# B&R Automation Studio project EasyLog
Automation Studio 4.12.3.127 SP; technology packages: mapp 5.24.1, mappCockpit 5.24.2, mappSafety 5.24.1, mappView 5.24.0

## Configuration C20

CPU 4PPC30.0702-21B, AutomationRuntime K4.93, Build 6.3.0, Safety 0.0, Vc V4.73.1

### Task classes (Cpu.sw)
```
Cyclic#2 (cycle 20000 us, tolerance 0 us):
  AsyncTask <- Async.AsyncTask.prg (AdditionalIncludeDirectories=\Logical\Async\AsyncCreation\ARM\, AdditionalLibraryDirectories=\Logical\Async\AsyncCreation\ARM\, AdditionalLibraries=AR)
  Example4 <- Example4.prg
Binaries: FWRules, arcoal, arsvcreg, TCData, arflatprv, mvLoader, udbdef, mCoWebSc, User, iomap, sysconf, Role, ashwd, arconfig, asfw, ashwac
Libraries: standard, runtime, astime, AsBrStr, sys_lib, ArEventLog, AsFifo, EasyLog, asiodiag, asioacc, SfDomDrv, SfDomVis, asepl, arssl, mpbase, MpSfDomMgr, aruser, fileio, asusb, astcp
```

### Hardware
```
4PPC30_0702_21B : 4PPC30.0702-21B v1.1.3.0
  Connector IF3:
    ActivateDevice = 1
    Mode = Manual
    InternetAddress = 10.10.10.100
    SubnetMask = 255.255.255.0
    InaPort = 11160
    ActivateSnmp = 2
  ConfigurationID = EasyLog_Config1
  TimerDeviceType = SWIOTIMER
  Cyclic1Duration = 10000
  Cyclic1Tolerance = 0
  Cyclic2Duration = 20000
  Cyclic2Tolerance = 0
  Cyclic3Duration = 50000
  Cyclic3Tolerance = 50000
  Cyclic4Duration = 100000
  Cyclic4Tolerance = 100000
  Cyclic5Duration = 200000
  Cyclic5Tolerance = 200000
  Cyclic6Duration = 500000
  Cyclic6Tolerance = 500000
  Cyclic7Duration = 1000000
  Cyclic7Tolerance = 1000000
  Cyclic7Stack = 65365
  Cyclic8Duration = 10000
  Cyclic8Tolerance = 30000000
  FileDevice1
  FileDeviceName1 = USER
  FileDevicePath1 = USER_PATH
  KeyMappingFile = VC\4PPC30_0702_21B1.dis
```

## Configuration Config1

CPU PC_any, AutomationRuntime I4.93, Build 6.3.0, Safety 0.0, Vc V4.73.1

### Task classes (Cpu.sw)
```
Cyclic#4:
  Program <- Program.prg
Binaries: FWRules, arcoal, arsvcreg, TCData, arflatprv, mvLoader, udbdef, mCoWebSc, User, iomap, sysconf, Role, ashwd, arconfig, asfw, ashwac
Libraries: AsIecCon, standard, runtime, astime, AsBrStr, DataObj, sys_lib, AsUSB, FileIO, AsSem, ArEventLog, AsARCfg, AsTCP, AsFifo, AsHttp, AsMem, EasyLog, asiodiag, asioacc, SfDomDrv, SfDomVis, asepl, arssl, mpbase, MpSfDomMgr, aruser
```

## Configuration ConfigNewC70

CPU 4PPC70.0573-20B, AutomationRuntime I4.93, Build 6.3.0, Vc V4.73.2

### Task classes (Cpu.sw)
```
Cyclic#2:
  Example4 <- Example4.prg
VcDataObjects: Visu1 <- Visu1.dob
Binaries: FWRules, arcoal, arsvcreg, TCData, arflatprv, mvLoader, udbdef, mCoWebSc, vcfile, arialbd, vcpdi855, vcbclass, vcnet, vcdsloc, Visu103, vccovl, vcptelo, vcshared, vcrt, vcpkat, vcpk, Visu101, vccbtn, vcmgr, Visu102, vctcal, vcalarm, vcpdsw, arial, vcgclass, vcpdvnc, vcpdihd, vcfntttf, vccstr, vcpdi815, vcpfppc7, vcdsint, User, iomap, sysconf, Role, ashwd, arconfig, asfw, ashwac
Libraries: EasyLog, AsBrStr, ArEventLog, astcp, asusb, astime, fileio, asiodiag, standard, asioacc, SfDomDrv, sys_lib, SfDomVis, asepl, runtime, arssl, mpbase, MpSfDomMgr, aruser, dataobj, vcresman
```

### Hardware
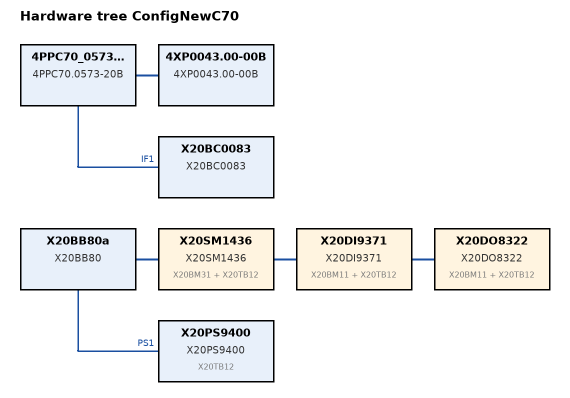
```
4PPC70_0573_20B : 4PPC70.0573-20B v1.5.4.0
  Connector IF2:
    ActivateDevice = 1
    Vnc1
    VncVcObjectName1 = Visu1
    VncKeyMappingFile1 = VC\PS2-Keyboard.dis
  ConfigurationID = EasyLog_ConfigNewC70
  UserPartitionSize = 0
  Cyclic1Tolerance = 0
  Cyclic2Tolerance = 0
  Cyclic7Stack = 65365
  FileDevice1
  FileDeviceName1 = USER
  FileDevicePath1 = USER_PATH
  VcObjectName = Visu1
  KeyMappingFile = VC\4PPC70_0573_20B.dis
4XP0043.00-00B : 4XP0043.00-00B v2.1.0.0  [X2X1 -> 4PPC70_0573_20B.IF5 [Cable Type=X2XCable, Length=10, Version=1.0.0.3]]
  Supervision = off
X20BB80a : X20BB80 v1.1.0.0
X20BC0083 : X20BC0083 v2.14.0.0  [PLK1 -> 4PPC70_0573_20B.IF1 (NodeNumber=1) [Cable Type=PowerlinkCable, Length=10, Version=1.0.0.3]; SL -> X20BB80a.SL1]
  Supervision = off
X20BM11a : X20BM11 v1.1.0.0  [X2X1 -> X20BM31a.X2X2]
X20BM11b : X20BM11 v1.1.0.0  [X2X1 -> X20BM11a.X2X2]
X20BM31a : X20BM31 v1.1.0.0  [X2X1 -> X20BB80a.IF1]
X20DI9371 : X20DI9371 v1.4.0.0  [SS1 -> X20TB12c.SS; SL -> X20BM11a.SL1]
  Supervision = off
X20DO8322 : X20DO8322 v1.5.0.0  [SS1 -> X20TB12d.SS; SL -> X20BM11b.SL1]
  Supervision = off
X20PS9400 : X20PS9400 v1.8.0.0  [SS1 -> X20TB12b.SS; PS -> X20BB80a.PS1]
  Supervision = off
X20SM1436 : X20SM1436 v2.3.0.0  [SS1 -> X20TB12a.SS; SL -> X20BM31a.SL1]
  FunctionModel = Standard
  Supervision = off
X20TB12a : X20TB12 v1.0.0.0
X20TB12b : X20TB12 v1.0.0.0
X20TB12c : X20TB12 v1.0.0.0
X20TB12d : X20TB12 v1.0.0.0
```

## Configuration Dinamic_Intel

CPU X20CP1686X, AutomationRuntime 6.0.2, Build 11.3.0, Vc 6.0.0

### Task classes (Cpu.sw)
```
Cyclic#4:
  Example1 <- Example1.prg
  Example2 <- Example2.prg
  Example3 <- Example3.prg
Libraries: EasyLog, runtime, ArEventLog, AsBrStr, sys_lib, standard
```

### Hardware
```
X20CP1686X : X20CP1686X v1.8.2.0
  FileDevice1
  FileDeviceName1 = USER
  FileDevicePath1 = USER_PATH
```

## Configuration Dynamic_ARM

CPU 4PPC30.043F-21B, AutomationRuntime 6.0.2, Build 11.3.0, Vc 6.0.0

### Task classes (Cpu.sw)
```
Cyclic#2 (cycle 20000 us, tolerance 20000 us):
  Example1 <- Example1.prg
  Example2 <- Example2.prg
  Example3 <- Example3.prg
Libraries: operator, runtime, AsIecCon, astime, EasyLog, ArEventLog, AsBrStr, sys_lib, standard
```

### Task classes (Cpu.sw)
```
Cyclic#3 (cycle 50000 us, tolerance 50000 us):
  Example2 <- Example2.prg
Cyclic#4 (cycle 100000 us, tolerance 100000 us):
  Example1 <- Example1.prg
Binaries: FWRules, TCData, mvLoader, udbdef, mCoWebSc, User, iomap, sysconf, Role, ashwd, arconfig, asfw, ashwac, arcoal, arsvcreg, arflatprv
Libraries: standard, runtime, EasyLog, asstring, astime, AsBrStr, sys_lib, ArEventLog, AsFifo, SfDomDrv, SfDomVis, MpSfDomMgr, AsIecCon, AsMem, DataObj, AsARCfg, AsSem, AsHttp
```

### Hardware
```
4PPC30_043F_21B : 4PPC30.043F-21B v1.1.4.0
  Connector IF3:
    ActivateDevice = 1
  ConfigurationID = EasyLog6_Dynamic_ARM
  TimerDeviceType = SWIOTIMER
  Cyclic1Duration = 10000
  Cyclic1Tolerance = 10000
  Cyclic2Duration = 20000
  Cyclic2Tolerance = 20000
  Cyclic3Duration = 50000
  Cyclic3Tolerance = 50000
  Cyclic4Duration = 100000
  Cyclic4Tolerance = 100000
  Cyclic5Duration = 200000
  Cyclic5Tolerance = 200000
  Cyclic6Duration = 500000
  Cyclic6Tolerance = 500000
  Cyclic7Duration = 1000000
  Cyclic7Tolerance = 1000000
  Cyclic8Duration = 10000
  Cyclic8Tolerance = 30000000
  FileDevice1
  FileDeviceName1 = USER
  FileDevicePath1 = USER_PATH
  KeyMappingFile = VC\4PPC30_043F_21B.dis
```

## Configuration Dynamic_ARM_2

CPU 4PPC30.043F-21B, AutomationRuntime K4.93, Build 6.3.0, Vc V4.73.2

### Task classes (Cpu.sw)
```
Cyclic#2 (cycle 20000 us, tolerance 20000 us):
  Example1 <- Example1.prg
  Example2 <- Example2.prg
  Example3 <- Example3.prg
Binaries: arsvcreg, udbdef, TCData, arflatprv, arcoal, mvLoader, FWRules, mCoWebSc, ashwac, User, sysconf, iomap, asfw, arconfig, ashwd, Role
Libraries: EasyLog, runtime, AsBrStr, sys_lib, ArEventLog, standard, astime, AsFifo, mpbase, arssl, SfDomVis, asiodiag, asioacc, aruser, fileio, SfDomDrv, asepl, MpSfDomMgr, asusb, astcp
```

### Hardware
```
4PPC30_043F_21B : 4PPC30.043F-21B v1.1.3.0
  Connector IF3:
    ActivateDevice = 1
  ConfigurationID = EasyLog_Dynamic_ARM_2
  TimerDeviceType = SWIOTIMER
  Cyclic1Duration = 10000
  Cyclic1Tolerance = 10000
  Cyclic2Duration = 20000
  Cyclic2Tolerance = 20000
  Cyclic3Duration = 50000
  Cyclic3Tolerance = 50000
  Cyclic4Duration = 100000
  Cyclic4Tolerance = 100000
  Cyclic5Duration = 200000
  Cyclic5Tolerance = 200000
  Cyclic6Duration = 500000
  Cyclic6Tolerance = 500000
  Cyclic7Duration = 1000000
  Cyclic7Tolerance = 1000000
  Cyclic8Duration = 10000
  Cyclic8Tolerance = 30000000
  FileDevice1
  FileDeviceName1 = USER
  FileDevicePath1 = USER_PATH
  KeyMappingFile = VC\4PPC30_043F_21B.dis
```

## Configuration Dynamic_Intel

CPU PC_any, AutomationRuntime K4.93, Build 6.3.0, Safety 0.0, Vc V4.73.1

CPU X20CP1586, AutomationRuntime H4.93, Build 6.3.0, Safety 0.0, Vc V4.73.1

### Task classes (Cpu.sw)
```
Cyclic#3:
  Example2 <- Example2.prg
Cyclic#4:
  Example1 <- Example1.prg
Binaries: FWRules, arcoal, arsvcreg, TCData, arflatprv, mvLoader, udbdef, mCoWebSc, User, iomap, sysconf, Role, ashwd, arconfig, asfw, ashwac
Libraries: standard, runtime, astime, AsBrStr, sys_lib, ArEventLog, AsFifo, asiodiag, asioacc, SfDomDrv, SfDomVis, asepl, arssl, mpbase, MpSfDomMgr, aruser, EasyLog, asstring
```

### Task classes (Cpu.sw)
```
Cyclic#2 (cycle 100000 us, tolerance 100000 us):
  Example1 <- Example1.prg
  Example2 <- Example2.prg
  Example3 <- Example3.prg
Binaries: FWRules, arcoal, arsvcreg, TCData, arflatprv, mvLoader, udbdef, mCoWebSc, User, iomap, sysconf, Role, ashwd, arconfig, asfw, ashwac
Libraries: standard, runtime, astime, AsBrStr, sys_lib, ArEventLog, AsFifo, EasyLog, asiodiag, asioacc, SfDomDrv, SfDomVis, asepl, arssl, mpbase, MpSfDomMgr, aruser, fileio, asusb, astcp
```

### Hardware
```
X20CP1586 : X20CP1586 v1.11.0.0
  Connector IF1:
    ActivateIna = 0
  Connector IF2:
    ActivateDevice = 1
    InaPort = 11160
  ConfigurationID = EasyLog_Config1
  Cyclic1Duration = 20000
  Cyclic1Tolerance = 0
  Cyclic1Stack = 522920
  Cyclic2Duration = 100000
  Cyclic2Tolerance = 100000
  FileDevice1
  FileDeviceName1 = USER
  FileDevicePath1 = USER_PATH
```

## Configuration ETA_Light

CPU 4PPC70.0573-20B, AutomationRuntime I4.93, Build 6.3.0, Safety 0.0, Vc V4.73.1

### Task classes (Cpu.sw)
```
Cyclic#2:
  Example4 <- Example4.prg
  AsyncTask <- Async.AsyncTask.prg (AdditionalIncludeDirectories=\Logical\Async\AsyncCreation\ARM\, AdditionalLibraryDirectories=\Logical\Async\AsyncCreation\ARM\, AdditionalLibraries=AR)
Binaries: FWRules, arcoal, arsvcreg, TCData, arflatprv, mvLoader, udbdef, mCoWebSc, User, iomap, sysconf, Role, ashwd, arconfig, asfw, ashwac
Libraries: standard, runtime, astime, AsBrStr, sys_lib, ArEventLog, AsFifo, EasyLog, asiodiag, asioacc, SfDomDrv, SfDomVis, asepl, arssl, mpbase, MpSfDomMgr, aruser, fileio, asusb, astcp
```

### Hardware
```
4PPC70_0573_20B : 4PPC70.0573-20B v1.5.4.0
  Connector IF2:
    ActivateDevice = 1
    Mode = Manual
    InternetAddress = 10.10.10.11
    SubnetMask = 255.255.255.0
    InaPort = 11160
    ActivateSnmp = 2
    DeviceParam = /EDDN=cpsw
  ConfigurationID = EasyLog_Config1
  Cyclic2Tolerance = 0
  Cyclic2Stack = 65365
  Cyclic7Stack = 65365
  FileDevice1
  FileDeviceName1 = USER
  FileDevicePath1 = USER_PATH
  KeyMappingFile = VC\4PPC70_0573_20B.dis
```

## Configuration Static_ARM

CPU X20CP0410, AutomationRuntime K4.93, Build 6.3.0, Safety 0.0, Vc V4.73.1

### Task classes (Cpu.sw)
```
Cyclic#3 (cycle 50000 us, tolerance 50000 us):
  Example2 <- Example2.prg
Cyclic#4 (cycle 100000 us, tolerance 100000 us):
  Example1 <- Example1.prg
Binaries: FWRules, arcoal, arsvcreg, TCData, arflatprv, mvLoader, udbdef, mCoWebSc, User, iomap, sysconf, Role, ashwd, arconfig, asfw, ashwac
Libraries: standard, runtime, astime, AsBrStr, sys_lib, ArEventLog, AsFifo, EasyLog, asiodiag, asioacc, SfDomDrv, SfDomVis, asepl, arssl, mpbase, MpSfDomMgr, aruser, AsIecCon, AsMem, DataObj, FileIO, AsARCfg, AsSem, AsHttp, AsUSB, AsTCP
```

### Hardware
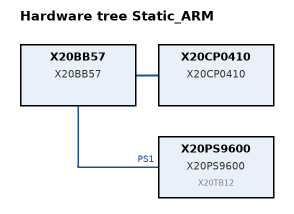
```
X20BB57 : X20BB57 v1.2.0.0
X20CP0410 : X20CP0410 v1.6.0.0  [SL -> X20BB57.SL1]
  Connector IF2:
    ActivateDevice = 1
    InaPort = 11160
  ConfigurationID = EasyLog_Config1
  TimerDeviceType = SWIOTIMER
  Cyclic1Duration = 10000
  Cyclic1Tolerance = 10000
  Cyclic2Duration = 20000
  Cyclic2Tolerance = 20000
  Cyclic3Duration = 50000
  Cyclic3Tolerance = 50000
  Cyclic4Duration = 100000
  Cyclic4Tolerance = 100000
  Cyclic5Duration = 200000
  Cyclic5Tolerance = 200000
  Cyclic6Duration = 500000
  Cyclic6Tolerance = 500000
  Cyclic7Duration = 1000000
  Cyclic7Tolerance = 1000000
  Cyclic8Duration = 10000
  Cyclic8Tolerance = 30000000
  FileDevice1
  FileDeviceName1 = USER
  FileDevicePath1 = USER_PATH
X20PS9600 : X20PS9600 v1.6.1.0  [PS -> X20BB57.PS1; SS1 -> X20TB12.SS]
X20TB12 : X20TB12 v1.0.0.0
```

## Configuration Static_Intel

CPU PC_any, AutomationRuntime K4.93, Build 6.3.0, Safety 0.0, Vc V4.73.1

### Task classes (Cpu.sw)
```
Cyclic#3:
  Example2 <- Example2.prg
Cyclic#4:
  Example1 <- Example1.prg
Binaries: FWRules, arcoal, arsvcreg, TCData, arflatprv, mvLoader, udbdef, mCoWebSc, User, iomap, sysconf, Role, ashwd, arconfig, asfw, ashwac
Libraries: standard, runtime, astime, AsBrStr, sys_lib, ArEventLog, AsFifo, EasyLog, asiodiag, asioacc, SfDomDrv, SfDomVis, asepl, arssl, mpbase, MpSfDomMgr, aruser
```

## Logical view

Binary libraries used (declarations not repeated): operator, runtime, AsIecCon, astime, ArEventLog, AsBrStr, sys_lib, standard, AsFifo

### Package Logical/Libraries - Global libraries

### Library Logical/Libraries/EasyLog (ANSIC, version 1.00.0)
Depends on: ArEventLog, AsBrStr, sys_lib

#### EasyLog.fun
```iecst
FUNCTION EasyLog : DINT (*Status returned by the function. Status <> ERR_OK should be checked*)
	VAR_INPUT
		Execute : BOOL; (*Input to add a message in the logger. Every cycle with TRUE in this input will insert a logger message. *) (* *) (*#PAR*)
		LoggerName : STRING[10]; (*String with the name of the Logger. Max Lenght 10 characters.*) (* *) (*#PAR*)
		LogLevel : USINT; (*Severity of the error. Coud be arEVENTLOG_SEVERITY_SUCCESS, arEVENTLOG_SEVERITY_INFO,  arEVENTLOG_SEVERITY_WARNING or arEVENTLOG_SEVERITY_ERROR*) (* *) (*#PAR*)
		ErrorNumber : UINT; (*Number of the error or information to insert*) (* *) (*#PAR*)
		Message : STRING[256]; (*String that specify the message to insert in the logger. Max lenght 256 characters*) (* *) (*#PAR*)
	END_VAR
END_FUNCTION
```

#### Logger.h
```c
#ifndef LOGGER_H
#define LOGGER_H

#include <stdlib.h>
#include "AsBrStr.h"
#include <cstring>
#include <string>

extern "C"
{
  long int EasyLog(plcbit Execute, plcstring* LoggerName, unsigned char LogLevel, unsigned short ErrorNumber, plcstring* Message);
}

#endif // LOGGER_H
```

#### EasyLog.cpp
```cpp
#include "Logger.h"
#include "EasyLog.h"
#include "LoggerInternal.hpp"

//extern "C" {
long int EasyLog(plcbit Execute, plcstring* LoggerName, unsigned char LogLevel, unsigned short ErrorNumber, plcstring* Message)
{
	Logger& logger = Logger::getInstance();
	return logger.EasyLogInternal(Execute, LoggerName, LogLevel, ErrorNumber, Message);
}
//}
```

#### LoggerInternal.hpp
```cpp
#ifndef LOGGERINTERNAL_H
#define LOGGERINTERNAL_H

#include "ArEventLog.h"
#include <stdlib.h>
#include "AsBrStr.h"
#include "runtime.h"
#include "sys_lib.h"
#include <iostream>
#include <cstring>
#include <string>
#include <queue>
#include <map>
#include "rtk.h"

struct LoggerEntry_type
{
	unsigned char LogLevel;
	long int ErrorNumber;
	char AsciiData[257];
};

struct LoggerHandler_type
{
	signed long ErrorInternal;
	char LoggerName[11];
	unsigned long pLoggerQueue;
	struct LoggerEntry_type LogEntry;
	unsigned long LogIdent;
	struct ArEventLogCreate ArEventLogCreate_0;
	RTK_TASK_H TaskHandler;
	bool CreatingLogger;
	bool CreateLogger;
};

class Logger {
public:
    static Logger& getInstance();
	long int EasyLogInternal(plcbit Execute, plcstring* LoggerName, unsigned char LogLevel, unsigned short ErrorNumber, plcstring* Message);

private:
    Logger() = default;
    ~Logger() = default;
    Logger(const Logger&) = delete;
    Logger& operator=(const Logger&) = delete;

	//Headers of the functions
    unsigned long SearchMap(unsigned long inst);
    long int UserLogEnqueue(unsigned char LogLevel, unsigned short ErrorNumber, unsigned long pAsciiData, unsigned long pLoggerName, unsigned long pHandler);
    long int UserLogWrite(unsigned long pHandler, bool fromAsync);
    long int UserLogCreateLog(unsigned long pHandler);
    long int UserLogGetIdent(unsigned long pHandler);
    static void CreateNewLoggerAsync(void* Params);

};

#endif // LOGGERINTERNAL_H
```

#### EasyLogInternal.cpp
```cpp
#include "LoggerInternal.hpp"
#include <cstdlib>
#include <cstring>

	/* Internal Data Map
	 * This map is used to store and retrieve the internal state for each instance, allowing
	 * for the management of multiple instances within the system. Related a Handler with all the information
	 * with one logger name given as a string */
std::map<std::string, unsigned long> internalMap;

	//Functions to get ident and write. As long as this functions have syncronous
	// execution does not have any sense save one copy of each function in the handler
struct ArEventLogGetIdent ArEventLogGetIdent_0;
struct ArEventLogWrite ArEventLogWrite_0;

Logger& Logger::getInstance() {
	static Logger instance;
	return instance;
}

/**
 * Retrieves or creates the internal data structure for the given instance.
 *
 * This function checks if an internal data structure for the provided instance
 * exists in the internal map. If it does not, it initializes a new internal
 * structure and stores it in the map.
 */
unsigned long Logger::SearchMap(unsigned long inst)
{
	//Retrieve the logger name
	std::string loggerName((char*)inst);
	std::map<std::string, unsigned long>::iterator it;

	//Search the Handler with the logger name
	it = internalMap.find(loggerName);

	//If it is not found, create a new Handler to insert to the map with the new logger name
	if (it == internalMap.end())
	{
		//Local instance of the handler
		struct LoggerHandler_type newHandler = {0};
		newHandler.LoggerName[11] = {0};
		std::strncpy(newHandler.LoggerName, loggerName.c_str(), sizeof(newHandler.LoggerName) - 1);

		//Create a local instance of queue, allocate it in memory and
		//achieve the pointer to that queue to store it in the local handler
		std::queue<LoggerEntry_type>* localLoggerQueue = (std::queue<LoggerEntry_type>*)malloc(sizeof(std::queue<LoggerEntry_type>));
		new(localLoggerQueue) std::queue<LoggerEntry_type>();
		newHandler.pLoggerQueue = reinterpret_cast<unsigned long>(localLoggerQueue);

		//Allocate the Handler in memory and save the local instance)
		LoggerHandler_type* savedInstance = (LoggerHandler_type*)malloc(sizeof(LoggerHandler_type));

		//Copy the local instance to the saved memory
		brsmemcpy((UDINT)savedInstance, (UDINT)&newHandler, sizeof(LoggerHandler_type));

		//Store the pointer of the saved instance
		unsigned long pHandler = reinterpret_cast<unsigned int>(savedInstance);

		//Save the new instance in the map and return it
		internalMap[loggerName] = pHandler;
		return internalMap[loggerName];
	}
	//If it is found return the Handler
	else
	{
		return it->second;
	}
}

/* Function to execute when is necessary a log insertion.
	It will be enqueued in a Queue until the UserLogWrite inserts the messages in the logger*/
long int Logger::UserLogEnqueue(unsigned char LogLevel, unsigned short ErrorNumber, unsigned long pAsciiData, unsigned long pLoggerName, unsigned long pHandler)
{
	//Initial status
	long int Status = ERR_OK;

	//Retrieve the Handler and its queue through its pointers
	struct LoggerHandler_type* Handler = reinterpret_cast<LoggerHandler_type*>(pHandler);
	std::queue<LoggerEntry_type>* queue = reinterpret_cast<std::queue<LoggerEntry_type>*>(Handler->pLoggerQueue);

	//Check not null pointers
	if (pHandler == 0 || Handler->pLoggerQueue == 0)
	{
		Status = ERR_BUR_ILLBPTR;
	}
	else
	{
		//Create a new entry type with the external information
		LoggerEntry_type newEntry;
		newEntry.LogLevel = LogLevel;
		newEntry.ErrorNumber = ErrorNumber;
		brsmemcpy((UDINT)&newEntry.AsciiData, pAsciiData, sizeof(newEntry.AsciiData));

		//Push that entry in the queue
		queue->push(newEntry);
	}

	return Status;
}

//Function to execute asyncronously with the Logger name to insert
// the messages in the logger that has been inserted with the UserLogEnqueue function
long int Logger::UserLogWrite(unsigned long pHandler, bool fromAsync)
{
	//Initialize the Status
	long int Status = ERR_OK;

	//Retrieve the Handler and its queue through its pointers
	struct LoggerHandler_type* Handler = reinterpret_cast<LoggerHandler_type*>(pHandler);
	std::queue<LoggerEntry_type>* queue = reinterpret_cast<std::queue<LoggerEntry_type>*>(Handler->pLoggerQueue);

	//Check not null pointers
	if (pHandler == 0 || Handler->pLoggerQueue == 0)
	{
		Status = ERR_BUR_ILLBPTR;
	}
	else
	{
		//If it is not busy the creation of the logger
		if (!Handler->CreatingLogger || fromAsync)
		{
			//Check if it is necessary to write the log
			if (queue->size() > 0 && Handler->LogIdent != 0)
			{
				int elements = queue->size();
				for (int i = 0; i < elements; i++)
				{
					// Put the first entry in the Handler
					Handler->LogEntry = queue->front();

					//Set the parameters of the write function
					ArEventLogWrite_0.Execute = 1;
					ArEventLogWrite_0.AddDataFormat = arEVENTLOG_ADDFORMAT_TEXT;
					ArEventLogWrite_0.AddDataSize = brsstrlen((UDINT)&Handler->LogEntry.AsciiData) + 1;
					ArEventLogWrite_0.AddData = (UDINT)&Handler->LogEntry.AsciiData;
					ArEventLogWrite_0.EventID = ArEventLogMakeEventID(Handler->LogEntry.LogLevel,0,Handler->LogEntry.ErrorNumber);
					brsstrcpy((UDINT)ArEventLogWrite_0.ObjectID, (UDINT)&Handler->LoggerName);
					ArEventLogWrite_0.Ident = Handler->LogIdent;
					ArEventLogWrite(&ArEventLogWrite_0);

					//Written OK. Quit from the queue and finish the process
					if (ArEventLogWrite_0.Done)
					{
						//Reset the function
						ArEventLogWrite_0.Execute = 0;
						ArEventLogWrite(&ArEventLogWrite_0);

						if (queue->size()>0)
						{
							//Delete the fist message
							queue->pop();
						}
					}
					//Error case
					else if (ArEventLogWrite_0.Error)
					{
						//Get the error
						Handler->ErrorInternal = Handler->ErrorInternal ? Handler->ErrorInternal : ArEventLogWrite_0.StatusID;
						Status = ArEventLogWrite_0.StatusID;

						//Reset the function
						ArEventLogWrite_0.Execute = 0;
						ArEventLogWrite(&ArEventLogWrite_0);
					}
				}
			}
		}
	}

	Handler->ErrorInternal = Status;

	return Status;
}

//Function to execute asyncronously to create a new logger if it does not exist
void Logger::CreateNewLoggerAsync(void *Params)
{
	// Recast Parameters to LoggerHandler_type*
	unsigned long  pHandler = reinterpret_cast<unsigned long>(Params);
	struct LoggerHandler_type* Handler = reinterpret_cast<LoggerHandler_type*>(pHandler);

	//Parameters of the new Logger
	Handler->ArEventLogCreate_0.Execute = 1;
	brsstrcpy((UDINT)&Handler->ArEventLogCreate_0.Name, (UDINT)&Handler->LoggerName);
	Handler->ArEventLogCreate_0.Size = 200000;
	Handler->ArEventLogCreate_0.Persistence = arEVENTLOG_PERSISTENCE_PERSIST;

	//Execute as many times it takes to finish, ok or with errors
	do
	{
	  ArEventLogCreate(&Handler->ArEventLogCreate_0);
	} while (Handler->ArEventLogCreate_0.Busy);

	//Created OK, Reset the create function and write the pending entries
	if (Handler->ArEventLogCreate_0.Done)
	{
		//Save the logger ident
		Handler->LogIdent = Handler->ArEventLogCreate_0.Ident;

		//Reset function
		Handler->ArEventLogCreate_0.Execute = 0;
		ArEventLogCreate(&Handler->ArEventLogCreate_0);

		//Write pending entries
		Logger::getInstance().UserLogWrite(pHandler, 1);
		Handler->CreatingLogger = 0;
	}

	//Error case. Reset the create function and inform the error
	else if (Handler->ArEventLogCreate_0.Error)
	{
		Handler->CreatingLogger = 0;

		//Get the error
		Handler->ErrorInternal = Handler->ErrorInternal ? Handler->ErrorInternal : Handler->ArEventLogCreate_0.StatusID;

		//Reset the function
		Handler->ArEventLogCreate_0.Execute = 0;
		ArEventLogCreate(&Handler->ArEventLogCreate_0);
	}

	//Delete this task once finished
	RtkDeleteTask(RtkGetCurrentTaskIdent());
}

long int Logger::UserLogCreateLog(unsigned long pHandler)
{
	//Initialize the Status
	long int Status = ERR_OK;

	//Retrieve the Handler through its pointer
	struct LoggerHandler_type* Handler = reinterpret_cast<LoggerHandler_type*>(pHandler);

	//Check not null pointers
	if (pHandler == 0)
	{
		Status = ERR_BUR_ILLBPTR;
	}
	else
	{
		if (!Handler->CreatingLogger)
		{
			//Launch the asyncronous task to create the logger if necessary
			if (Handler->CreateLogger && Handler->CreatingLogger == 0)
			{
				Handler->CreatingLogger = 1;
				LPRTK_CREATE_TASK_FKT function = &CreateNewLoggerAsync;
				const char* taskName =  Handler->LoggerName;
				void* pHandlerVoid = reinterpret_cast<void*>(pHandler);
				RtkCreateTask(taskName, 10, 0x1000, 0x1000, RTK_TASK_RESUMED, function, pHandlerVoid, &Handler->TaskHandler);
			}
		}
	}
	return Status;
}

//Function to execute asyncronously with the Logger name to insert
// the messages in the logger that has been inserted with the UserLogEnqueue function
long int Logger::UserLogGetIdent(unsigned long pHandler)
{
	//Initialize the Status
	long int Status = ERR_OK;

	//Retrieve the Handler and its queue through its pointers
	struct LoggerHandler_type* Handler = reinterpret_cast<LoggerHandler_type*>(pHandler);

	//Check not null pointers
	if (pHandler == 0)
	{
		Status = ERR_BUR_ILLBPTR;
	}
	else
	{
		Handler->CreateLogger = 0;
		//Only search the logger if the log ident does not exist
		if (Handler->LogIdent == 0)
		{
			//If it is not busy the creation of the logger
			if (!Handler->CreatingLogger)
			{
				//Get the info log
				ArEventLogGetIdent_0.Execute = 1;
				brsstrcpy((UDINT)ArEventLogGetIdent_0.Name, (UDINT)&Handler->LoggerName);
				ArEventLogGetIdent(&ArEventLogGetIdent_0);

				//Finded the logger
				if (ArEventLogGetIdent_0.Done)
				{
					//Save the logger ident in the handler
					Handler->LogIdent = ArEventLogGetIdent_0.Ident;

					//Reset the function
					ArEventLogGetIdent_0.Execute = 0;
					ArEventLogGetIdent(&ArEventLogGetIdent_0);
				}
					//First appearing of the logger, necessary creation
				else if (ArEventLogGetIdent_0.StatusID == arEVENTLOG_ERR_LOGBOOK_NOT_FOUND)
				{
					//Flag to star the creation of the logger
					Handler->CreateLogger = 1;

					//Reset the function
					ArEventLogGetIdent_0.Execute = 0;
					ArEventLogGetIdent(&ArEventLogGetIdent_0);
				}
				//Error case
				else if (ArEventLogGetIdent_0.Error)
				{
					Handler->ErrorInternal = Handler->ErrorInternal ? Handler->ErrorInternal : ArEventLogGetIdent_0.StatusID;

					//Get the error
					Status = ArEventLogGetIdent_0.StatusID;

					//Reset the function
					ArEventLogGetIdent_0.Execute = 0;
					ArEventLogGetIdent(&ArEventLogGetIdent_0);
				}
			}
		}
	}
	return Status;
}

/* Function to insert messages in custom loggers in an aeasy way. The Executed is detected by Edge*/
long int Logger::EasyLogInternal(plcbit Execute, plcstring* LoggerName, unsigned char LogLevel, unsigned short ErrorNumber, plcstring* Message)
{
	//Initialize the different status
	long int Status = ERR_OK;
	long int StatusEnqueue = ERR_OK;
	long int StatusGetIdent = ERR_OK;
	long int StatusWrite = ERR_OK;

	//Get the pointer to the logger name
	char* pCharMessage = Message;
	unsigned long pMessage = reinterpret_cast<unsigned long>(pCharMessage);

	//Get the pointer to the message
	char* pCharLoggerName = LoggerName;
	unsigned long pLoggerName = reinterpret_cast<unsigned long>(pCharLoggerName);

	//Search the handler in the map
	unsigned long pHandler = SearchMap(pLoggerName);

	//Command to insert a new message
	if (Execute)
	{
		//Check that the parameters are correct when an insertion is needed
		if (strcmp(Message, "") == 0 || strcmp(LoggerName, "") == 0 || LogLevel < 0 || LogLevel > 3)
		{
			//Wrong parameters
			Status = ERR_BUR_ILLPAR;
		}
		else
		{
			//Enqueue the message in the Queue
			StatusEnqueue = UserLogEnqueue(LogLevel, ErrorNumber, pMessage, pLoggerName, pHandler);
		}
	}

	//Write the pending messages (or create the logger in the first insertion)
	if (strcmp(LoggerName, "") != 0)
	{
		StatusGetIdent = UserLogGetIdent(pHandler);
		UserLogCreateLog(pHandler);
		StatusWrite = UserLogWrite(pHandler, 0);
	}
	else
	{
		//Necessary logger name
		Status = ERR_BUR_ILLPAR;
	}

	//Check the errors
	if (Status == ERR_OK)
	{
		if (StatusEnqueue != ERR_OK)
		{
			Status = StatusEnqueue;
		}
		if (StatusGetIdent != ERR_OK)
		{
			Status = StatusGetIdent;
		}
		if(StatusWrite != ERR_OK)
		{
			Status = StatusWrite;
		}
	}

	return Status;
}
```

#### heap.cpp - Dynamic memory allocation reserve
```cpp
unsigned long bur_heap_size = 0x3FFFC; //256 KB
```

#### rtkTimer.h
```c
/**
 * @file
 * @brief RTK timer functions
 *
 * Timers can be used for cyclic actions and for single timeouts
 *
 * @ingroup rtk
 */

#ifndef _RTK_TIMER_H_
#define _RTK_TIMER_H_

#include <rtkBase.h>

#ifdef __cplusplus
extern "C" {
#endif

/** @brief RTK timer handle */
typedef RTK_H RTK_TIMER_H;

/** @brief Type of RTK timer flags */
typedef unsigned long RTK_TIMERFLAG;

/** @name Flags for RtkStartTimer() */
/*@{*/
#define RTK_TIMER_CYCLIC 0x00000000
#define RTK_TIMER_ONESHOT 0x00000001
/*@}*/

/**
 * @brief Create a timer object with the provided name ('lpszTimerName' must be unique or NULL).
 *
 * When the timer expires (to be started with RtkStartTimer()), then timerFunction(timerContext) is called with task
 * priority 'wTimerPriority' and with stack size 'ulTimerSupervidorStackSize'.
 * The output-parameter 'hTimer' (must not be NULL) returns a handle to the timer. */
EXIMPORT RTK_ERROR RtkCreateTimer(const char* lpszTimerName, WORD wTimerPriority, ULONG ulTimerSupervisorStackSize,
                                  LPRTK_CREATE_TASK_FKT timerFunction, void* timerContext, RTK_TIMER_H* hTimer);

/** @brief Deletes a timer object */
EXIMPORT RTK_ERROR RtkDeleteTimer(RTK_TIMER_H hTimer);

/**
 * @brief Starts a cyclical timer ('TimerFlags'=RTK_TIMER_CYCLIC) with the provided cycle time ('ulTimerCycleUsec')
 * or a single-shot timer ('TimerFlags'=RTK_TIMER_ONESHOT) with the provided delay ('ulTimerCycleUsec') */
EXIMPORT RTK_ERROR RtkStartTimer(RTK_TIMER_H hTimer, ULONG ulTimerCycleUsec, RTK_TIMERFLAG TimerFlags);

/** @brief Stops a timer started with RtkStartTimer() */
EXIMPORT RTK_ERROR RtkStopTimer(RTK_TIMER_H hTimer);

#ifdef __cplusplus
}
#endif

#endif
```

#### rtkRtc.h
```c
/**
 * @file
 * @brief Functions to set and read the real-time-clock
 * @ingroup rtk
 */

#ifndef _RTK_RTC_H_
#define _RTK_RTC_H_

#include <rtkBase.h>

#ifdef __cplusplus
extern "C" {
#endif

/**
 * @brief  Set the real-time-clock to 'newDateTime'.
 *
 *  'newDateTime' has to contain the localtime (not the UTC time). */
EXIMPORT RTK_ERROR RtkSetRealTimeClock(RTK_RTC const* newDateTime);

/** @brief Retrieves the current date and localtime. */
EXIMPORT void RtkGetRealTimeClock(RTK_RTC* dateTime);

#if AR_CORE
#include "private/rtkRtcP.h"
#endif

#ifdef __cplusplus
}
#endif

#endif
```

#### rtkTypes.h
```c
/**
 * @file
 * @brief Contains legacy type definitions.
 * @note These types should only be used for calling functions which require these types.
 * @ingroup rtk
 */

#ifndef _RTK_TYPES_H_
#define _RTK_TYPES_H_

#include <stdint.h>

#ifdef __cplusplus
extern "C" {
#endif

#ifndef TRUE
#define TRUE 1
#define FALSE 0
#endif

/** @cond */
#ifndef _ULONG_DEFINED_ /* ULONG might also be defined by vxTypesOld.h */
#define _ULONG_DEFINED_
/** @endcond */
typedef uint32_t ULONG;
#endif

/** @cond */
#ifndef _BYTE_DEFINED_ /* BYTE might already be defined from plctypes.h */
#define _BYTE_DEFINED_
/** @endcond */
typedef uint8_t BYTE;
#endif

/** @cond */
#ifndef _WORD_DEFINED_ /* WORD might already be defined from plctypes.h */
#define _WORD_DEFINED_
/** @endcond */
typedef uint16_t WORD;
#endif

typedef unsigned char BOOLEAN;
typedef char* LPSTRING;
typedef void* LPVOID;
typedef BYTE* LPBYTE;
typedef WORD* LPWORD;
typedef ULONG* LPULONG;

/** @brief RTK type of realtime clock */
typedef struct
{
	WORD Year;        /**< @brief 0 up (for example 1999)		*/
	BYTE Month;       /**< @brief 1-12							*/
	BYTE Day;         /**< @brief 1-31							*/
	BYTE DayOfWeek;   /**< @brief 1=monday, ..., 7=sunday		*/
	BYTE Hour;        /**< @brief 0-23							*/
	BYTE Minute;      /**< @brief 0-59							*/
	BYTE Second;      /**< @brief 0-59							*/
	WORD Millisecond; /**< @brief 0-999							*/
	WORD Microsecond; /**< @brief 0-999							*/
} RTK_RTC, *LPRTK_RTC;

#ifdef __cplusplus
}
#endif

#endif
```

#### EasyLog.typ - not listed in the package file held
```iecst
TYPE
	InputsEasyLogTyp : 	STRUCT
		LogLevel : USINT; (*Severity of the error. Coud be arEVENTLOG_SEVERITY_SUCCESS, arEVENTLOG_SEVERITY_INFO,  arEVENTLOG_SEVERITY_WARNING or arEVENTLOG_SEVERITY_ERROR*)
		ErrorNumber : UINT; (*Number of the error or information to insert*)
		Message : STRING[256]; (*String that specify the message to insert in the logger. Max lenght 256 characters*)
		LoggerName : STRING[10]; (*String with the name of the Logger. Max Lenght 10 characters*)
	END_STRUCT;
END_TYPE
```

#### EasyLog.var - not listed in the package file held
```iecst
(*********************************************************************
 * Logger Constants
 ********************************************************************)
VAR CONSTANT
	MAX_LOGGER_QUEUE : USINT := 10;
END_VAR
```

#### GlobalIncludes.h - not listed in the package file held
```c
#include "rtk.h"
/* Datatypes and datatypes of function blocks */
typedef enum LoggerStep_enum
{	LOGGER_WAIT,
	LOGGER_GET_INFO_LOG,
	LOGGER_CREATE_LOG,
	LOGGER_WRITE
} LoggerStep_enum;

typedef struct LoggerEntry_type
	{
	unsigned char LogLevel;
	long int ErrorNumber;
	char AsciiData[257];
} LoggerEntry_type;

typedef struct LoggerFifo_type
	{
	unsigned char PendingEntries;
	struct LoggerEntry_type Entry[20];
} LoggerFifo_type;

typedef struct LoggerHandler_type
	{	signed long ErrorInternal;
	char LoggerName[11];
	enum LoggerStep_enum LogStep;
	struct LoggerFifo_type LogFifo;
	struct LoggerEntry_type LogEntry;
	unsigned long LogIdent;
	struct ArEventLogGetIdent ArEventLogGetIdent_0;
	struct ArEventLogCreate ArEventLogCreate_0;
	struct ArEventLogWrite ArEventLogWrite_0;
	plcbit LastExecute;
	RTK_TASK_H TaskHandler;
} LoggerHandler_type;
```

#### GlobalIncludes.hpp - not listed in the package file held
```cpp
#include "rtk.h"
#include <queue>

/* Datatypes and datatypes of function blocks */
typedef struct LoggerEntry_type
	{
	unsigned char LogLevel;
	long int ErrorNumber;
	char AsciiData[257];
} LoggerEntry_type;

typedef struct LoggerHandler_type
	{	signed long ErrorInternal;
	char LoggerName[11];
	unsigned long pLoggerQueue;
	struct LoggerEntry_type LogEntry;
	unsigned long LogIdent;
	struct ArEventLogCreate ArEventLogCreate_0;
	RTK_TASK_H TaskHandler;
	bool CreatingLogger;
	bool CreateLogger;
} LoggerHandler_type;
```

#### EasyLog.c - not listed in the package file held
```c
#include <bur/plctypes.h>
#ifdef __cplusplus
	extern "C"
	{
#endif
	#include "EasyLog.h"
#ifdef __cplusplus
	};
#endif
/* Function to insert messager in custom loggers in an aeasy way */
signed long EasyLog(plcbit Execute, struct InputsEasyLogTyp* LoggerInfo)
{
	/*TODO: Add your code here*/
}
```

#### UserLogWrite.cpp - not listed in the package file held
```cpp
#include <bur/plctypes.h>
#ifdef __cplusplus
	extern "C"
	{
#endif
#include "EasyLog.h"
#include "GlobalIncludes.h"
#ifdef __cplusplus
	};
#endif

#include "ArEventLog.h"
#include <stdlib.h>
#include "AsBrStr.h"
#include "runtime.h"
#include "sys_lib.h"
#include <iostream>
#include <cstring>
#include <string>
#include <map>
#include "rtk.h"

#define sdRB_ERR_ASSERT 1001

/**
 * Internal Data Map
 *
 * This map is used to store and retrieve the internal state for each instance, allowing
 * for the management of multiple instances within the system. Related a Handler with all the information
with one logger name given as a string
 */
static std::map<std::string, struct LoggerHandler_type> internalMap;

long int UserLogWrite(struct LoggerHandler_type* Handler);

static bool creatingLogger;

/**
 * Retrieves or creates the internal data structure for the given instance.
 *
 * This function checks if an internal data structure for the provided instance
 * exists in the internal map. If it does not, it initializes a new internal
 * structure and stores it in the map.
 */
struct LoggerHandler_type* SearchMap(unsigned long inst){

	std::string loggerName((char*)inst);
	std::map<std::string, struct LoggerHandler_type>::iterator it;

	//Search the Handler with the logger name
	it = internalMap.find(loggerName);

	//If it is not found, create a new Handler to insert to the map with the new logger name
	if (it == internalMap.end())
	{
		struct LoggerHandler_type newHandler = {0};
		newHandler.LoggerName[11] = {0};
		std::strncpy(newHandler.LoggerName, loggerName.c_str(), sizeof(newHandler.LoggerName) - 1);
		internalMap[loggerName] = newHandler;
		return &internalMap[loggerName];
	}
		//If it is fount return the Handler
	else
	{
		return &it->second;
	}
}

/* Function to execute when is necessary a log insertion.
	It will be enqueued in a Fifo until the UserLogWrite inserts the messages in the logger*/
long int UserLogEnqueue(unsigned char LogLevel, unsigned short ErrorNumber, unsigned long pAsciiData, unsigned long pLoggerName, struct LoggerHandler_type* Handler)
{

	long int Status = ERR_OK;

	if (Handler->LogFifo.PendingEntries < sizeof(Handler->LogFifo.Entry) / sizeof(Handler->LogFifo.Entry[0]) - 1) {
		Handler->LogFifo.Entry[Handler->LogFifo.PendingEntries].LogLevel = LogLevel;
		Handler->LogFifo.Entry[Handler->LogFifo.PendingEntries].ErrorNumber = ErrorNumber;
		brsmemcpy((UDINT)&Handler->LogFifo.Entry[Handler->LogFifo.PendingEntries].AsciiData, pAsciiData, sizeof(Handler->LogFifo.Entry[Handler->LogFifo.PendingEntries].AsciiData));
		if (brsstrlen((UDINT)&Handler->LogFifo.Entry[Handler->LogFifo.PendingEntries].AsciiData) >= sizeof(Handler->LogFifo.Entry[Handler->LogFifo.PendingEntries].AsciiData)) {
			brsstrcpy((UDINT)&Handler->LogFifo.Entry[Handler->LogFifo.PendingEntries].AsciiData + sizeof(Handler->LogFifo.Entry[Handler->LogFifo.PendingEntries].AsciiData) - 4, (UDINT)&"...");
		}
		Handler->LogFifo.PendingEntries++;
	}
	else if (Handler->LogFifo.PendingEntries < sizeof(Handler->LogFifo.Entry) / sizeof(Handler->LogFifo.Entry[0])) {
		Status = ERR_FUB_BUSY;
	}
	return Status;
}

//Function to execute asyncronously to create a new logger if it does not exist
void CreateNewLoggerAsync(void *Params)
{

	// Recast Parameters to LoggerHandler_type*
	LoggerHandler_type* Handler = static_cast<LoggerHandler_type*>(Params);

	//Status = ERR_FUB_BUSY;
	//Parameters of the new Logger
	Handler->ArEventLogCreate_0.Execute = 1;
	brsstrcpy((UDINT)&Handler->ArEventLogCreate_0.Name, (UDINT)&Handler->LoggerName);
	Handler->ArEventLogCreate_0.Size = 200000;
	Handler->ArEventLogCreate_0.Persistence = arEVENTLOG_PERSISTENCE_PERSIST;

	do
	{
	  ArEventLogCreate(&Handler->ArEventLogCreate_0);
	} while (!Handler->ArEventLogCreate_0.Done && !Handler->ArEventLogCreate_0.Error);

	//Finished LogCreate. Move forward
	if (Handler->ArEventLogCreate_0.Done)
	{
		Handler->ArEventLogCreate_0.Execute = 0;
		Handler->LogIdent = Handler->ArEventLogCreate_0.Ident;
		ArEventLogCreate(&Handler->ArEventLogCreate_0);

		creatingLogger = 0;
		//Once created, call the function to insert the pending entries
		//UserLogWrite(Handler);

	}
		//Error case
	else if (Handler->ArEventLogCreate_0.Error)
	{

		creatingLogger = 0;
		Handler->ArEventLogCreate_0.Execute = 0;
		Handler->ErrorInternal = Handler->ErrorInternal ? Handler->ErrorInternal : Handler->ArEventLogCreate_0.StatusID;
		//Status = Handler->ArEventLogCreate_0.StatusID;
		ArEventLogCreate(&Handler->ArEventLogCreate_0);

	}

	//Delete the task once finished
	RtkDeleteTask(RtkGetCurrentTaskIdent());

}

//Function to execute asyncronously with the Logger name to insert
// the messages in the logger that has been inserted with the UserLogEnqueue function
long int UserLogGetIdent(struct LoggerHandler_type* Handler)
{

	//Initialize the Status
	long int Status = ERR_OK;
	Handler->CreateLogger = 0;
	Handler->WriteEntries = 0;
	//If it is not busy the creation of the logger
	if (!creatingLogger)
	{
		// Put the first entry in the Handler
		Handler->LogEntry = Handler->LogFifo.Entry[0];

		//Get the info log
		Handler->ArEventLogGetIdent_0.Execute = 1;
		brsstrcpy((UDINT)&Handler->ArEventLogGetIdent_0.Name, (UDINT)&Handler->LoggerName);
		ArEventLogGetIdent(&Handler->ArEventLogGetIdent_0);

		//Finished getIdent, move forward
		if (Handler->ArEventLogGetIdent_0.Done)
		{
			Handler->ArEventLogGetIdent_0.Execute = 0;
			Handler->LogIdent = Handler->ArEventLogGetIdent_0.Ident;
			ArEventLogGetIdent(&Handler->ArEventLogGetIdent_0);
			if (Handler->LogFifo.PendingEntries > 0)
			{
				Handler->WriteEntries = 1;
				Status = ERR_FUB_BUSY;
			}
			else
			{
				Status = ERR_OK;
			}
		}
			//First appearing of the logger, necessary creation
		else if (Handler->ArEventLogGetIdent_0.StatusID == arEVENTLOG_ERR_LOGBOOK_NOT_FOUND)
		{
			Handler->ArEventLogGetIdent_0.Execute = 0;
			Handler->CreateLogger = 1;
			ArEventLogGetIdent(&Handler->ArEventLogGetIdent_0);
			Status = ERR_FUB_BUSY;
		}
			//Error case
		else if (Handler->ArEventLogGetIdent_0.Error)
		{
			Handler->ArEventLogGetIdent_0.Execute = 0;
			Handler->ErrorInternal = Handler->ErrorInternal ? Handler->ErrorInternal : Handler->ArEventLogGetIdent_0.StatusID;
			ArEventLogGetIdent(&Handler->ArEventLogGetIdent_0);
			Status = Handler->ArEventLogGetIdent_0.StatusID;
		}
	}
	return Status;
}

long int UserLogCreateLog(struct LoggerHandler_type* Handler)
{
	//Initialize the Status
	long int Status = ERR_OK;
	if (!creatingLogger)
	{
		//Launch the asyncronous task to create the logger
		if (Handler->CreateLogger && creatingLogger == 0)
		{
			creatingLogger = 1;
			LPRTK_CREATE_TASK_FKT function = &CreateNewLoggerAsync;
			const char* taskName =  Handler->LoggerName;
			RtkCreateTask(taskName, 10, 0x1000, 0x1000, RTK_TASK_RESUMED, function, Handler, &Handler->TaskHandler);
		}
	}

	return Status;
}

//Function to execute asyncronously with the Logger name to insert
// the messages in the logger that has been inserted with the UserLogEnqueue function
long int UserLogWrite(struct LoggerHandler_type* Handler)
{
	//Initialize the Status
	long int Status = ERR_OK;
	Handler->ErrorInternal = ERR_OK;

	// Local temporary variables which are used in many places
	UDINT i;

	//If it is not busy the creation of the logger
	if (!creatingLogger)
	{
		//Check if it is necessary to write the log
		if (Handler->WriteEntries && Handler->LogFifo.PendingEntries > 0)
		{
			for (int i = 0; i < Handler->LogFifo.PendingEntries; i++)
			{
				Status = ERR_FUB_BUSY;
				Handler->ArEventLogWrite_0.Execute = 1;
				Handler->ArEventLogWrite_0.AddDataFormat = arEVENTLOG_ADDFORMAT_TEXT;
				Handler->ArEventLogWrite_0.AddDataSize = brsstrlen((UDINT)&Handler->LogEntry.AsciiData) + 1;
				Handler->ArEventLogWrite_0.AddData = (UDINT)&Handler->LogEntry.AsciiData;
				Handler->ArEventLogWrite_0.EventID = ArEventLogMakeEventID(Handler->LogEntry.LogLevel,0,Handler->LogEntry.ErrorNumber);
				brsstrcpy((UDINT)&Handler->ArEventLogWrite_0.ObjectID, (UDINT)&Handler->LoggerName);
				Handler->ArEventLogWrite_0.Ident = Handler->LogIdent;
				ArEventLogWrite(&Handler->ArEventLogWrite_0);

				//Written OK. Quit from the queue and finish the process
				if (Handler->ArEventLogWrite_0.Done)
				{
					Handler->ArEventLogWrite_0.Execute = 0;
					ArEventLogWrite(&Handler->ArEventLogWrite_0);

					//Quit the entry of the Fifo once is writted
					for (i = 0; i < (UDINT)Handler->LogFifo.PendingEntries - 1; i++)
					{
						Handler->LogFifo.Entry[i] = Handler->LogFifo.Entry[i+1];
					}
					brsmemset((UDINT)&Handler->LogFifo.Entry[Handler->LogFifo.PendingEntries-1], 0 , sizeof(Handler->LogFifo.Entry[0]));
					Handler->LogFifo.PendingEntries--;

					Status = ERR_OK;
				}
					//Error case
				else if (Handler->ArEventLogWrite_0.Error)
				{
					Handler->ArEventLogWrite_0.Execute = 0;
					Handler->ErrorInternal = Handler->ErrorInternal ? Handler->ErrorInternal : Handler->ArEventLogWrite_0.StatusID;
					Status = Handler->ArEventLogWrite_0.StatusID;
					ArEventLogWrite(&Handler->ArEventLogWrite_0);
				}
			}
		}
	}

	Handler->ErrorInternal = Status;

	return Status;
}

/* Function to insert messages in custom loggers in an aeasy way. The Executed is detected by Edge*/
long int EasyLog(plcbit Execute, plcstring* LoggerName, unsigned char LogLevel, unsigned short ErrorNumber, plcstring* Message)
{
	//Initialize the different status
	long int Status = ERR_OK;
	long int StatusEnqueue = ERR_OK;
	long int StatusWrite = ERR_OK;

	//Get the pointer to the logger name
	char* pCharMessage = Message;
	unsigned long pMessage = reinterpret_cast<unsigned long>(pCharMessage);

	//Get the pointer to the message
	char* pCharLoggerName = LoggerName;
	unsigned long pLoggerName = reinterpret_cast<unsigned long>(pCharLoggerName);

	//Search the map to check the last execute
	struct LoggerHandler_type* Handler = SearchMap(pLoggerName);

	//Command to insert a new message
	if (Execute)
	{
		//Check that the parameters are correct when an insertion is needed
		if (strcmp(Message, "") == 0 || strcmp(LoggerName, "") == 0 || LogLevel < 0 || LogLevel > 3)
		{
			Status = ERR_BUR_ILLPAR;
		}
		else
		{
			//Enqueue the message in the Fifo
			StatusEnqueue = UserLogEnqueue(LogLevel, ErrorNumber, pMessage, pLoggerName, Handler);
		}
	}

	//Write the pending messages (or create the logger in the first insertion)
	if (strcmp(LoggerName, "") != 0)
	{
		UserLogGetIdent(Handler);
		UserLogCreateLog(Handler);
		StatusWrite = UserLogWrite(Handler);
	}
	else
	{
		Status = ERR_BUR_ILLPAR;
	}

	//Check the errors
	if (Status == ERR_OK)
	{
		if (StatusEnqueue != ERR_OK)
		{
			Status = StatusEnqueue;
		}
		if(StatusWrite != ERR_OK)
		{
			Status = StatusWrite;
		}
	}

	return Status;
}
```

### Program Logical/Example1 (IEC)

#### Variables.var
```iecst
VAR
	Message : STRING[256];
	Status : DINT;
	Temperature : INT;
	TempStr : STRING[80];
	InsertMessages : BOOL;
END_VAR
```

#### Main.st
```iecst
(*********************************************************************************
 * Copyright: B&R Industrial Automation GmbH
*********************************************************************************
 * Program: Example3
 * File: Example 3 - EasyLogLibrary
 * Author:    B&R Spain
 * Created:   November 18, 2024/10:04 AM
*********************************************************************************
 * Description: Example to show how to insert cyclicaly the value of a variable
	in a logger
 * Interface:
	-
*************************** VERSION CONTROL *************************************
   Version	| Date	                | Author	| Description
----------------------------------------------------------------------------------
   V1.00	| November 18, 2024		| B&R Spain	|  Initial version
 *********************************************************************************)

PROGRAM _INIT
	// Set an initial message
	Message := 'TestMessage';

	//This will create the logger in case that does not exist in advance.
	//This is only necessary if the insert time will be very fast < 5ms.
	// In that case this call with FALSE in Execute will create the logger to avoid Cycle Time Violation
	Status := EasyLog(FALSE, 'Temp', arEVENTLOG_SEVERITY_INFO, 123,  Message);

END_PROGRAM

PROGRAM _CYCLIC

    // Convert the current temperature into a string
	brsitoa(Temperature, ADR(TempStr));
	TempStr := CONCAT(TempStr, ' şC');
	Message := CONCAT('Current Temperature: ', TempStr);

	// Execute the logger insertion if InsertMessages = TRUE
	Status := EasyLog(InsertMessages, 'Temp', arEVENTLOG_SEVERITY_INFO, 123,  Message);

	IF Status <> ERR_OK THEN
		//Check the error in the help and solve it
	END_IF;

END_PROGRAM

PROGRAM _EXIT

END_PROGRAM
```

### Program Logical/Example2 (IEC)

#### Variables.var
```iecst
VAR
	Message : STRING[256];
	Status : DINT;
	Temperature : INT;
	AlarmLimit : INT := 40;
	WarningLimit : INT := 30;
	TempStr : STRING[80];
	AlarmLimitStr : STRING[80];
	WarningLimitStr : STRING[80];
	TemperatureAlarm : BOOL;
	TemperatureWarning : BOOL;
END_VAR
```

#### Main.st
```iecst
(*********************************************************************************
 * Copyright: B&R Industrial Automation GmbH
*********************************************************************************
 * Program: Example2
 * File: Example 2 - EasyLogLibrary
 * Author:    B&R Spain
 * Created:   November 18, 2024/10:04 AM
*********************************************************************************
 * Description: Example to show how to insert alarms in a logger
	-
 * Interface:
	-
*************************** VERSION CONTROL *************************************
   Version	| Date	                | Author	| Description
----------------------------------------------------------------------------------
   V1.00	| November 18, 2024		| B&R Spain	|  Initial version
 *********************************************************************************)

PROGRAM _INIT

END_PROGRAM

PROGRAM _CYCLIC

	// Convert the current temperature into a string
	brsitoa(Temperature, ADR(TempStr));
	TempStr := CONCAT(TempStr, ' şC');

	(********************************** ALARM LIMIT  **********************************)
	// Check if it is greater than the Alarm Limit and create the message
	IF Temperature > AlarmLimit THEN
		//Creation of the Message
		Message := CONCAT('Current Temperature: ', TempStr);
		Message := CONCAT(Message, ' above the Alarm limit: ');
		brsitoa(AlarmLimit, ADR(AlarmLimitStr));
		AlarmLimitStr := CONCAT(AlarmLimitStr, ' şC');
		Message := CONCAT(Message, AlarmLimitStr);
		TemperatureAlarm := TRUE;
	ELSE;
		TemperatureAlarm := FALSE;
	END_IF;

	//Make the call to the function with EDGEPOS to make only 1 insertion when the alarm raises
	Status := EasyLog(EDGEPOS(TemperatureAlarm), 'TempAlarm', arEVENTLOG_SEVERITY_ERROR, 1111,  Message);

	IF Status <> ERR_OK THEN
		//Check the error and solve it
	END_IF;

	(********************************** WARNING LIMIT  **********************************)
	// Check if it is greater than the Warning Limit and create the message
	IF Temperature > WarningLimit THEN
		//Creation of the Message
		Message := CONCAT('Current Temperature: ', TempStr);
		Message := CONCAT(Message, ' above the Warning limit: ');
		brsitoa(WarningLimit, ADR(WarningLimitStr));
		WarningLimitStr := CONCAT(WarningLimitStr, ' şC');
		Message := CONCAT(Message, WarningLimitStr);
		TemperatureWarning := TRUE;
	ELSE;
		TemperatureWarning := FALSE;
	END_IF;

	//Make the call to the function with EDGEPOS to make only 1 insertion when the warning raise
	Status := EasyLog(EDGEPOS(TemperatureWarning), 'TempAlarm', arEVENTLOG_SEVERITY_WARNING, 2222,  Message);

	IF Status <> ERR_OK THEN
		//Check the error and solve it
	END_IF;

END_PROGRAM

PROGRAM _EXIT
	(* Insert code here *)

END_PROGRAM
```

### Program Logical/Example3 (IEC)

#### Types.typ
```iecst
TYPE
	RecipeType : 	STRUCT
		Name : STRING[80];
		MaxTemp : INT;
	END_STRUCT;
END_TYPE
```

#### Variables.var
```iecst
VAR
	Message : STRING[256];
	Status : DINT;
	Recipe : RecipeType;
	RecipeOld : RecipeType;
	AuxStr : STRING[80];
END_VAR
```

#### Main.st
```iecst
(*********************************************************************************
 * Copyright: B&R Industrial Automation GmbH
*********************************************************************************
 * Program: Example3
 * File: Example 3 - EasyLogLibrary
 * Author:    B&R Spain
 * Created:   November 18, 2024/10:04 AM
*********************************************************************************
 * Description: Example to show how to insert changes in a recipe in the logger
	-
 * Interface:
	-
*************************** VERSION CONTROL *************************************
   Version	| Date	                | Author	| Description
----------------------------------------------------------------------------------
   V1.00	| November 18, 2024		| B&R Spain	|  Initial version
 *********************************************************************************)

PROGRAM _INIT
	//Set the initial Values of the Recipe
	Recipe.MaxTemp := 50;
	Recipe.Name := 'Recipe1';

	//Copy the initial value to the Old Recipe
	brsmemcpy(ADR(RecipeOld), ADR(Recipe), SIZEOF(Recipe));

END_PROGRAM

PROGRAM _CYCLIC

	(**********************************  Parameter: Name  **********************************)
	// Compare if the recipe name has changed
	IF 	brsmemcmp(ADR(RecipeOld.Name), ADR(Recipe.Name), SIZEOF(Recipe.Name)) <> 0 THEN
		//Creation of the message
		Message := CONCAT('Parameter Name of the recipe has changed. Old value = ', RecipeOld.Name);
		Message := CONCAT(Message, '. New value = ');
		Message := CONCAT(Message, Recipe.Name);

		//Register the change
		Status := EasyLog(TRUE, 'RcpChanges', arEVENTLOG_SEVERITY_INFO, 123,  Message);

		IF Status <> ERR_OK THEN
			//Check the error and solve it
		END_IF;

		//Save the new value
		RecipeOld.Name := Recipe.Name;
	END_IF;

	(**********************************  Parameter: MaxTemp  **********************************)
	// Compare if the recipe max temperature has changed
	IF 	brsmemcmp(ADR(RecipeOld.MaxTemp), ADR(Recipe.MaxTemp), SIZEOF(Recipe.MaxTemp)) <> 0 THEN
		//Creation of the message
		brsitoa(RecipeOld.MaxTemp, ADR(AuxStr));
		Message := CONCAT('Parameter MaxTemp of the recipe has changed. Old value = ', AuxStr);
		Message := CONCAT(Message, '. New value = ');
		brsitoa(Recipe.MaxTemp, ADR(AuxStr));
		Message := CONCAT(Message, AuxStr);

		//Register the change
		Status := EasyLog(TRUE, 'RcpChanges', arEVENTLOG_SEVERITY_INFO, 123,  Message);

		IF Status <> ERR_OK THEN
			//Check the error and solve it
		END_IF;

		//Save the new value
		RecipeOld.MaxTemp := Recipe.MaxTemp;
	END_IF;

END_PROGRAM

PROGRAM _EXIT
	(* Insert code here *)

END_PROGRAM
```

### Program Logical/Async/AsyncTask (ANSIC)

#### Main.cpp - Init, cyclic, exit code
```cpp
#include <bur/plctypes.h>

#ifdef _DEFAULT_INCLUDES
#include <AsDefault.h>
#endif
#include "rtk.h"

RTK_TASK_H TaskHandler1;
RTK_TASK_H TaskHandler2;

// amount of memory to be allocated for heap storage must be specified for every ANSI C++ program with the bur_heap_size variable
unsigned long bur_heap_size = 0xFFFF;

//Function to execute asyncronously to increase the value of the counter
void IncreaseCounter(void *Params)
{
	counter++;
	//Delete the task once finished
	RtkDeleteTask(RtkGetCurrentTaskIdent());
}

void _INIT ProgramInit(void)
{
	// Insert code here

}

void _CYCLIC ProgramCyclic(void)
{
	if (equalExecutes)
	{
		Execute2 = Execute1;
	}
	// Insert code here
	//Launch the asyncronous task to create the logger
	if (Execute1)
	{
		Execute1 = 0;
		LPRTK_CREATE_TASK_FKT function = &IncreaseCounter;
		RtkCreateTask(nullptr, 10, 0x1000, 0x1000, RTK_TASK_RESUMED, function, nullptr, &TaskHandler1);
	}

	if (Execute2)
	{
		Execute2 = 0;
		LPRTK_CREATE_TASK_FKT function = &IncreaseCounter;
		RtkCreateTask(nullptr, 10, 0x1000, 0x1000, RTK_TASK_RESUMED, function, nullptr, &TaskHandler2);
	}

}

void _EXIT ProgramExit(void)
{
	// Insert code here

}
```

#### Variables.var - Local variables
```iecst
VAR
	counter : DINT;
	equalExecutes : BOOL;
	Execute2 : BOOL;
	Execute1 : BOOL;
END_VAR
```

### rLib.h
```c
/**
 * @file
 * @brief The API provides functions for communicating with the second CPU of a redundant CPU pair.
 *
 * This API provides functionality for synchronous and asynchronous data exchange
 * between a redundant CPU pair connected via rLink.
 * The Data exchange is organized in communication channels with unique name identifier.
 * A communication channel is capable of sending and receiving asynchronous data on demand,
 * as well as copying a contiguous memory block synchronously with every cyclic taskclass execution.
 *
 * @ingroup rcpu
 */
#ifndef _RLIB_H_
#define _RLIB_H_

#include <stdint.h>

#ifdef __cplusplus
extern "C" {
#endif

/**
 * @brief The handle referring to a communication channel.
 */
typedef int32_t RLIB_H;

/**
 * @brief Open a communication channel for data transport in redundancy context.
 * @param name The unique name identifying the communication channel to be used on primary and secondary CPU.
 * @param size The payload size in bytes mandatory for synchronous data exchange (optional).
 * @param tx The memory address of producer (optional).
 * @param rx The memory address of consumer (optional).
 *
 * If all optional parameters are set, the source data provided by the producer is copied
 * to the destination memory of the consumer on every cycle of the calling task class.
 *
 * @returns The handle of the opened communication channel.
 */
RLIB_H rOpen(const char* name, uint32_t size, const void* tx, void* rx);

/**
 * @brief Close dedicated communication channel.
 * @param handle The handle of the communication channel.
 */
void rClose(RLIB_H handle);

/**
 * @brief Receive data by reading from the communication channel.
 * @param handle The handle of the communication channel.
 * @param buffer The destination buffer for the data to be read.
 * @param bytes The size in bytes of the destination buffer.
 *
 * @returns -1 on error, else the amount of bytes that could be read.
 */
int32_t rRead(RLIB_H handle, void* buffer, uint32_t bytes);

/**
 * @brief Send data by writing it to the communication channel.
 * @param handle The handle of the communication channel.
 * @param buffer The source buffer for data to be written.
 * @param bytes The size in bytes of the source buffer.
 *
 * @returns -1 on error, else the amount of bytes that could be written.
 */
int32_t rWrite(RLIB_H handle, const void* buffer, uint32_t bytes);

#ifdef __cplusplus
}
#endif

#endif
```

### rtkTask.h
```c
/**
 * @file
 * @brief RTK task functions
 * @ingroup rtk
 */

#ifndef _RTK_TASK_H_
#define _RTK_TASK_H_

#include <rtkBase.h>

#ifdef __cplusplus
extern "C"
{
#endif

/** @brief RTK task handle */
typedef RTK_H RTK_TASK_H;

/** @brief RTK task timer handle */
typedef RTK_H RTK_TASK_TIMER_H;

/** @name Miscellaneous task macros */
/*@{*/
#define RTK_TASKIDENT_ITSELF 0x00000000
#define RTK_MAX_TASK_PRIORITY 255
#define RTK_MIN_TASK_PRIORITY 1
#define RTK_IDLE_TASK_PRIORITY 0x1000
#define RTK_MAX_TASK_VALUES 16
/*@}*/

/** @brief Type of task flags */
typedef unsigned long RTK_TASKFLAG;

/** @name Task flags (create/start) */
/*@{*/
#define RTK_TASK_RESUMED 0x00000000 /**< @brief task starts immediately */
#define RTK_TASK_SUSPENDED 0x00000001 /**< @brief task does not start immediately (to be started with RtkTaskResume()) */
#define RTK_TASK_SYSTEM 0x00000000 /**< @brief ignored */
#define RTK_TASK_DRIVER 0x00000002 /**< @brief ignored */
#define RTK_TASK_APPLICATION 0x00000004 /**< @brief ignored */
/*@}*/

/** @name Priority classes
 *
 * We use priority classes to define the real-time requirements of a task.
 * A task of a certain class will not be interrupted by tasks of a lower class.
 * But the task may be interrupted by other tasks of the same class,
 * so that all tasks of the same class get evenly access to a CPU. */
/*@{*/

/**
 * @brief A task of this class has real-time requirements.
 *
 * This class should be chosen,
 * if the task generates a response to an other system. A task of this class is expected
 * to wake up at most every 1ms and consumes very little CPU Power.
 */
#define RTK_TASK_REALTIME_1MS 0x00000008

/**
 * @brief A task of this class has some kind of real-time requirements.
 *
 * This class should be chosen, if the task generates a response to a user or to an other system.
 * A task of this class is expected to wake up at most every 10ms and consumes little CPU Power.
 */
#define RTK_TASK_REALTIME_10MS 0x00000010

/**
 * @brief A task of this class has no real-time requirement.
 *
 * This class should be chosen, if some background calculations are performed.
 */
#define RTK_TASK_BEST_EFFORT 0x00000020
/*@}*/

/** @brief Type of task event flags */
typedef unsigned long RTK_EVENTFLAG;

/** @name Task event flags */
/*@{*/
#define RTK_EVENT_ANY 0x00000000       /**< @brief wait until any of the wanted events are set */
#define RTK_EVENT_ALL 0x00000001       /**< @brief wait until all wanted events are set */
#define RTK_EVENT_NO_DELETE 0x00000002 /**< @brief ignored */
/*@}*/

/** @brief Type of task state flags */
typedef unsigned long RTK_TASKSTATEFLAG;

/** @name Task state flags (taskInfo)
 * | combination of task state flags | |
 * |:-|:-
 * |(RTK_TASKSTATE_DELAYED + RTK_TASKSTATE_SUSPENDED)| Task is both delayed and suspended
 * |(RTK_TASKSTATE_PENDED  + RTK_TASKSTATE_SUSPENDED)| Task is both pended and suspended */
/*@{*/
#define RTK_TASKSTATE_READY 0x00000000     /**< @brief Task is not waiting for any resource other than the CPU. */
#define RTK_TASKSTATE_SUSPENDED 0x00000001 /**< @brief Task is unavailable for execution. */
#define RTK_TASKSTATE_PENDED 0x00000002    /**< @brief Task is blocked due to the unavailability of some resource. */
#define RTK_TASKSTATE_DELAYED 0x00000004   /**< @brief Task is asleep for some duration. */
/*@}*/

/**
 * @brief Creates a task running function 'taskFunction'('taskFunctionParameter').
 *
 * The task has the name 'lpszTaskName' (must be unique or NULL, please also note the behaviour if the maximum length
 * #MAX_RTK_NAME_LENGTH is exceeded), the priority 'wTaskPriority' (1.. lowest, 255.. highest), and the stack size
 * 'ulTaskUserStackSize' + 'ulTaskSupervisorStackSize' in bytes. This combined stack size has to be greater or equal to
 * 0x1000 and less than or equal to 0x100000, otherwise the error #ERR_RTK_NO_STACK will be returned. The 'TaskFlags'
 * can be used to determine the initial task state (resumed/suspended). The function returns a handle to the created
 * task ('hTask') */
EXIMPORT RTK_ERROR RtkCreateTask(const char* lpszTaskName, WORD wTaskPriority, ULONG ulTaskSupervisorStackSize,
                                 ULONG ulTaskUserStackSize, RTK_TASKFLAG TaskFlags, LPRTK_CREATE_TASK_FKT taskFunction,
                                 void* taskFunctionParameter, RTK_TASK_H* hTask);

/**
 * @brief Deletes the task.
 *
 * Stops execution and frees stack of the task. */
EXIMPORT RTK_ERROR RtkDeleteTask(RTK_TASK_H hTask);

/**
 * @brief Suspends the task.
 *
 * A suspended task stops its execution until it is resumed (RtkResumeTask()) */
EXIMPORT RTK_ERROR RtkSuspendTask(RTK_TASK_H hTask);

/** @brief Resumes the task. */
EXIMPORT RTK_ERROR RtkResumeTask(RTK_TASK_H hTask);

/** @brief Delays the calling task for the specified time in us. */
EXIMPORT void RtkSleepTaskUsec(ULONG ulSleepUsec);

/**
 * @brief Sends an event to a task ('hTask').
 *
 * Each bit of 'wTaskEvent' is one event of the task - sending multiple events is possible (logical OR of event-bits).
 * Sending one event-bit multiple times (e.g. by calling this function twice) has no effect if the event was not yet
 * read with RtkReceiveTaskEvent(). */
EXIMPORT RTK_ERROR RtkSendTaskEvent(RTK_TASK_H hTask, WORD wTaskEvents);

/**
 * @brief Waits for one ('EventFlags'=#RTK_EVENT_ANY) or all ('EventFlag'=#RTK_EVENT_ALL) of the requested
 * Events and returns these events. Resets all returned events of the task.
 * @param hTask            Handle of the task for which the events shall be returned
 * @param wWantedEvents    Bit-mask of the events which shall be returned
 * @param EventFlags       With 'EventFlags'=#RTK_EVENT_ANY this function returns if any of the events specified with
 *                         'wWantedEvents' is received. With 'EventFlags'=#RTK_EVENT_ALL this function only returns if
 * all of the events specified with 'wWantedEvents' is received.
 * @param ulTimeoutUsec    If the specified timeout is over before the events are received, the function returns with an
 *                         error and 'lpwReceivedEvent' is not valid. If some of the requested events were already
 * received by the task, then these events are not reset.
 * @param lpwReceivedEvent This output-parameter contains the received events after the function call.
 *                         Parameter must not be NULL. */
EXIMPORT RTK_ERROR RtkReceiveTaskEvent(RTK_TASK_H hTask, WORD wWantedEvents, RTK_EVENTFLAG EventFlags,
                                       ULONG ulTimeoutUsec, WORD* lpwReceivedEvents);

/**
 * @brief Cyclically sends events to a task ('hTask').
 *
 * The events will be sent every 'ulDelayUsec' us.
 * Each bit of 'wTaskEvent' is one event of the task - sending multiple events is possible (logical OR of event-bits)
 * Sending one event-bit multiple times has no effect (e.g. if the timer expires and the event is re-sent before the
 * event was read with RtkReceiveTaskEvent()).
 * Returns a timer handle ('hTaskTimer' - must not be NULL) which can be used to stop sending the events
 * (RtkCancelTaskTimer()) */
EXIMPORT RTK_ERROR RtkSendTaskEventCyclic(RTK_TASK_H hTask, WORD wTaskEvents, ULONG ulDelayUsec,
                                          RTK_TASK_TIMER_H* hTaskTimer);

/**
 * @brief Sends events once to a task ('hTask').
 *
 * The events will be sent after 'ulDelayUsec' us.
 * Each bit of 'wTaskEvent' is one event of the task - sending multiple events is possible (logical OR of event-bits).
 * Sending one event-bit multiple times (e.g. by calling this function twice) has no effect if the event was not yet
 * read with RtkReceiveTaskEvent().
 * Returns a timer handle ('hTaskTimer' - must not be NULL) which can be used to stop sending the event
 * (RtkCancelTaskTimer()) */
EXIMPORT RTK_ERROR RtkSendTaskEventAfter(RTK_TASK_H hTask, WORD wTaskEvents, ULONG ulDelayUsec,
                                         RTK_TASK_TIMER_H* hTaskTimer);

/**
 * @brief Cancels the provided timer ('hTaskTimer').
 *
 * This results in canceling sending the events initiated with RtkSendTaskEventCyclic() or RtkSendTaskEventAfter() */
EXIMPORT RTK_ERROR RtkCancelTaskTimer(RTK_TASK_TIMER_H hTaskTimer);

/**
 * @brief Writes to one of the 16 available local variables of the task ('hTask').
 *
 * 'byValueIndex' (0-15) addresses the variables, 'ulValue' is the values to be written */
EXIMPORT RTK_ERROR RtkSetTaskValue(RTK_TASK_H hTask, BYTE byValueIndex, ULONG ulValue);

/**
 * @brief Reads to one of the 16 available local variables of the task ('hTask').
 *
 * 'byValueIndex' (0-15) addresses the variables, 'lpulValue' contains the value of the variable after the function call
 */
EXIMPORT RTK_ERROR RtkGetTaskValue(RTK_TASK_H hTask, BYTE byValueIndex, ULONG* lpulValue);

/** @brief Sets the task priority to 'wTaskPriority' (1.. lowest, 255.. highest) */
EXIMPORT RTK_ERROR RtkSetTaskPriority(RTK_TASK_H hTask, WORD wTaskPriority);

/**
 * @brief Retrieves the task priority.
 *
 * 'lpwTaskPriority' contains the priority of the task after the function call */
EXIMPORT RTK_ERROR RtkGetTaskPriority(RTK_TASK_H hTask, WORD* lpwTaskPriority);

/**
 * @brief Returns task information.
 *
 * @param hTask              Handle of the task for which the information shall be returned
 * @param lpTaskStateFlags   Output-parameter - can be NULL. Returns the task state (RTK_TASKSTATE_READY,
 *                           RTK_TASKSTATE_SUSPENDED, RTK_TASKSTATE_PENDED, RTK_TASKSTATE_DELAYED)
 * @param lpwTaskPriority    Output-parameter - can be NULL. Returns the task priority
 * @param lpulUnused1        unused - can be NULL
 * @param lpulUnused2        unused - can be NULL
 * @param lpulFreeStack      Output-parameter - can be NULL. Returns the free stack size
 * @param pInternalTaskIdent Output-parameter - can be NULL. Returns an OS-specific task ident */
EXIMPORT RTK_ERROR RtkGetTaskInfo(RTK_TASK_H hTask, RTK_TASKSTATEFLAG* lpTaskStateFlags, WORD* lpwTaskPriority,
                                  ULONG* lpulUnused1, ULONG* lpulUnused2, ULONG* lpulFreeStack,
                                  void** pInternalTaskIdent);

/** @brief Get the handle for the currently running task */
EXIMPORT RTK_TASK_H RtkGetCurrentTaskIdent(void);

/** @returns TRUE if the task is ready, FALSE if the task is not ready or if 'hTask' is invalid. */
EXIMPORT BOOLEAN RtkIsTaskReady(RTK_TASK_H hTask);

/** @returns TRUE if the task is suspended, FALSE if the task is not suspended or if 'hTask' is invalid. */
EXIMPORT BOOLEAN RtkIsTaskSuspended(RTK_TASK_H hTask);

#ifdef __cplusplus
}
#endif

#endif
```

### rtk.h
```c
/**
 * @file
 * @brief This API provides abstractions for OS-functionalities (semaphores, tasks, timers, ...).
 *
 * Instead of using native Windows or VxWorks functions, you should use this API.
 * All functions returning RTK_ERROR return ERR_OK on success and other error codes on failure.
 *
 * @ingroup rtk
 */

#ifndef _RTK_H_
#define _RTK_H_

#include <rtkBase.h>
#include <rtkTask.h>
#include <rtkCriticalSection.h>
#include <rtkSemaphore.h>
#include <rtkMemory.h>
#include <rtkTimer.h>
#include <rtkFifo.h>
#include <rtkPlainFifo.h>
#include <rtkRtc.h>
#include <rtkObject.h>
#include <rtkMisc.h>

#if AR_CORE
#include <private/rtkP.h>
#endif

#endif
```

### Program Logical/Example4

#### Variables.var
```iecst
VAR
	Message : STRING[256];
	Status : DINT;
	AuxStr : STRING[80];
	i : UINT := 0;
	MessagesPerCycle : UINT := 2;
	InsertMessages4 : BOOL;
	InsertMessages3 : BOOL;
	InsertMessages2 : BOOL;
	InsertMessages : BOOL;
	LoggerName2 : STRING[10] := 'Log1_2';
	LoggerName : STRING[10] := 'Log1';
	OldLoggerName : STRING[10];
	MessageIndex : DINT;
	createInNextCycle : BOOL;
	createNewLogger : BOOL;
	BothInserts : BOOL;
	LoggerName3 : STRING[256];
	LoggerName4 : STRING[256];
	OneInsert : BOOL;
END_VAR
```

#### Main.st
```iecst
PROGRAM _INIT
	(* Set an initial message *)
	Message := 'TestMessage';

	//Repeat until finish the process, with or without errors
	// This will create the logger if it does not exist
//	REPEAT
//		Status := EasyLog(FALSE, LoggerName, arEVENTLOG_SEVERITY_INFO, 123,  Message);
//		UNTIL Status <> ERR_FUB_BUSY
//	END_REPEAT;

END_PROGRAM

PROGRAM _CYCLIC

	IF brsmemcmp(ADR(OldLoggerName), ADR(LoggerName), SIZEOF(LoggerName)) <> 0 THEN
		MessageIndex := 0;
		brsmemcpy(ADR(OldLoggerName), ADR(LoggerName), SIZEOF(LoggerName));
		brsmemcpy(ADR(LoggerName2), ADR(LoggerName), SIZEOF(LoggerName));
		LoggerName2 := CONCAT(LoggerName2, '2');
		brsmemcpy(ADR(LoggerName3), ADR(LoggerName), SIZEOF(LoggerName));
		LoggerName3 := CONCAT(LoggerName3, '3');
		brsmemcpy(ADR(LoggerName4), ADR(LoggerName), SIZEOF(LoggerName));
		LoggerName4 := CONCAT(LoggerName4, '4');

		InsertMessages := TRUE;
		InsertMessages2 := TRUE;
		InsertMessages3 := TRUE;
		InsertMessages4 := TRUE;
	END_IF;

	FOR i := 1 TO MessagesPerCycle DO
		//Message index inserted in this logger
		brsitoa(MessageIndex, ADR(AuxStr));
		MessageIndex := MessageIndex + 1;

		Message := CONCAT('Index = ', AuxStr);
		brsitoa(i, ADR(AuxStr));
		//Creation of the message
		Message := CONCAT(Message,' .Message number ');
		Message := CONCAT(Message, AuxStr);
		Message := CONCAT(Message, ' from   ');
		brsitoa(MessagesPerCycle, ADR(AuxStr));
		Message := CONCAT(Message, AuxStr);
		Message := CONCAT(Message, ' inserted this cycle ');
		//Register the change

		IF BothInserts THEN
			InsertMessages := TRUE;
			InsertMessages2 := TRUE;
			InsertMessages3 := TRUE;
			InsertMessages4 := TRUE;
		END_IF;

		IF InsertMessages THEN
			Status := EasyLog(InsertMessages, LoggerName, arEVENTLOG_SEVERITY_INFO, 123,  Message);
			IF OneInsert THEN
				InsertMessages := FALSE;
			END_IF;
		END_IF;
		IF InsertMessages2 THEN
			Status := EasyLog(InsertMessages2, LoggerName2, arEVENTLOG_SEVERITY_INFO, 123,  Message);
			//	InsertMessages2 := FALSE;
			IF OneInsert THEN
				InsertMessages2 := FALSE;
			END_IF;
		END_IF;

		IF InsertMessages3 THEN
			Status := EasyLog(InsertMessages3, LoggerName3, arEVENTLOG_SEVERITY_INFO, 123,  Message);
			//			InsertMessages3 := FALSE;
			IF OneInsert THEN
				InsertMessages3 := FALSE;
			END_IF;
		END_IF;

		IF InsertMessages4 THEN
			Status := EasyLog(InsertMessages4, LoggerName4, arEVENTLOG_SEVERITY_INFO, 123,  Message);
			//			InsertMessages4 := FALSE;
			IF OneInsert THEN
				InsertMessages4 := FALSE;
			END_IF;
		END_IF;

		BothInserts := FALSE;

	//	Status := EasyLog(InsertMessages2, LoggerName2, arEVENTLOG_SEVERITY_INFO, 123,  Message);

		IF MessageIndex >=200 THEN
			InsertMessages := FALSE;
			InsertMessages2 := FALSE;
			InsertMessages3 := FALSE;
			InsertMessages4 := FALSE;
		END_IF;

		IF Status <> ERR_OK AND Status <> ERR_FUB_BUSY THEN
			//Check the error and solve it
		END_IF;
	END_FOR;

	//	InsertMessages := FALSE;

END_PROGRAM

PROGRAM _EXIT
	(* Insert code here *)

END_PROGRAM
```

### Program Logical/FunAsync (ANSIC)

#### Cyclic.c - Cyclic code
```c
#include <bur/plctypes.h>

#ifdef _DEFAULT_INCLUDES
	#include <AsDefault.h>
#endif

#include <stdio.h>
#include "rtk.h"

void myAsynchronousFunction(void)
{
	do
	{
	  Counter++;
	} while (Block);
	RtkDeleteTask(RtkGetCurrentTaskIdent());
}

void _CYCLIC ProgramCyclic(void)
{
	if (Cmd[0])
	{
		Cmd[0] = 0;
		LPRTK_CREATE_TASK_FKT function = (LPRTK_CREATE_TASK_FKT)&myAsynchronousFunction;
		RTK_TASK_H hTask;
		RtkCreateTask(NULL, 50, 0x1000, 0x1000, 0, function, NULL, &hTask);
	} else if (Cmd[1])
	{
		Cmd[1] = 0;
		LPRTK_CREATE_TASK_FKT function = (LPRTK_CREATE_TASK_FKT)&myAsynchronousFunction;
		RTK_TASK_H hTask0;
		RTK_TASK_H hTask1;
		RtkCreateTask(NULL, 50, 0x1000, 0x1000, 0, function, NULL, &hTask0);
		RtkCreateTask(NULL, 50, 0x1000, 0x1000, 0, function, NULL, &hTask1);
	}
}
```

#### Variables.var - Local variables
```iecst
VAR
	Counter : DINT := 0;
	Cmd : ARRAY[0..1] OF BOOL;
	Block : BOOL;
END_VAR
```

#### rtkObject.h
```c
/**
 * @file
 * @brief Functions to read general information about RTK objects
 * @ingroup rtk
 */

#ifndef _RTK_OBJECT_H_
#define _RTK_OBJECT_H_

#include <rtkBase.h>

#ifdef __cplusplus
extern "C" {
#endif

/** @name RTK object types */
/*@{*/
typedef enum
{
	RTK_OBJ_INVALID = 0,
	RTK_OBJ_TASK,
	RTK_OBJ_SEMAPHORE,
	RTK_OBJ_CRITICAL_SECTION,
	RTK_OBJ_TIMER,
	RTK_OBJ_INTERRUPT,
	RTK_OBJ_EXCEPTION,
	RTK_OBJ_PLAINFIFO,
	RTK_OBJ_FIFO,
	RTK_OBJ_MEMORY,
	RTK_OBJ_SHARED_MEMORY,
	RTK_OBJ_DEBUGGER,
	RTK_OBJ_LOG,
	RTK_OBJ_RTC,
	RTK_OBJ_MISC,
	RTK_OBJ_TASKTIMER /* internal */
} RTK_OBJ_TYPE;
/*@}*/

/** @brief RTK object type pointer */
typedef RTK_OBJ_TYPE* LPRTK_OBJ_TYPE;

/**
 * @brief Searches an RTK object with the provided name ('lpszObjectName').
 *
 * Returns the object ('hObject' - must not be NULL) and the type of the object ('lpObjectType' - can be NULL) */
EXIMPORT RTK_ERROR RtkGetIdent(const char* lpszObjectName, RTK_H* hObject, LPRTK_OBJ_TYPE lpObjectType);

/**
 * @brief Returns information about the RTK-Object.
 * @param hObject         Handle of the RTK Object
 * @param ulMaxNameLength Length of the provided 'lpszObjectName' buffer
 * @param lpObjectType    Output-parameter - can be NULL. Returns the type of the RTK-object.
 * @param lpszObjectName  Output-parameter - can be NULL. The function call writes the RTK-object name to this buffer */
EXIMPORT RTK_ERROR
RtkGetObjectInfo(RTK_H hObject, ULONG ulMaxNameLength, LPRTK_OBJ_TYPE lpObjectType, char* lpszObjectName);

#ifdef __cplusplus
}
#endif

#endif
```

#### rtkPlainFifo.h
```c
/**
 * @file
 * @brief RTK Plain FIFO
 *
 * Rtk plain FIFO is a simple ringbuffer which does not use any locking.
 * It is possible to have one task reading and one task writing to the FIFO without requiring any further locking.
 * If multiple tasks read or if multiple tasks write to the FIFO, then external locking is required.
 *
 * @ingroup rtk
 */

#ifndef _RTK_PLAIN_FIFO_H_
#define _RTK_PLAIN_FIFO_H_

#include <rtkBase.h>

#ifdef __cplusplus
extern "C" {
#endif

/** @brief RTK plain FIFO handle */
typedef RTK_H RTK_PLAIN_FIFO_H;

/**
 * @brief Creates a FIFO with the provided name ('lpszFifoName' must be unique or NULL).
 *
 * The FIFO provides space for 'ulFifoMaxEntries' with 'ulFifoEntrySize'.
 * A handle to the FIFO is returned as output-parameter ('hFifo' - must not be NULL) */
EXIMPORT RTK_ERROR
RtkCreatePlainFifo(const char* lpszFifoName, ULONG ulFifoEntrySize, ULONG ulFifoMaxEntries, RTK_PLAIN_FIFO_H* hFifo);

/** @brief Deletes a plain FIFO */
EXIMPORT RTK_ERROR RtkDeletePlainFifo(RTK_PLAIN_FIFO_H hFifo);

/**
 * @brief Writes data to the FIFO.
 *
 * The size of the data is the size provided with 'ulFifoEntrySize' when creating the FIFO. If the FIFO is full (it only
 * contains entries which were not yet read), then this function returns #ERR_RTK_FIFO_WRITE */
EXIMPORT RTK_ERROR RtkWritePlainFifo(RTK_PLAIN_FIFO_H hFifo, const void* lpDataSource);

/**
 * @brief Copies data from the FIFO to 'lpDataDestination' (must not be NULL).
 *
 * The size of the copied data is the size provided with 'ulFifoEntrySize' when creating the  FIFO.
 * @returns #ERR_RTK_FIFO_READ if the FIFO is empty */
EXIMPORT RTK_ERROR RtkReadPlainFifo(RTK_PLAIN_FIFO_H hFifo, void* lpDataDestination);

/**
 * @brief Deletes all data contained in the FIFO.
 *
 * This function requires external locking if another task calls RtkReadPlainFifo() */
EXIMPORT RTK_ERROR RtkClearPlainFifo(RTK_PLAIN_FIFO_H hFifo);

/**
 * @brief Obtains information about the FIFO.
 * @param hFifo Handle to the FIFO for which the information shall be retrieved
 * @param lpulFifoFree Output-parameter - can be NULL. Returns the amount of free FIFO entries
 * @param lpulFifoUsed Output-parameter - can be NULL. Returns the amount of occupied FIFO entries
 * @param lpulFifoEntrySize Output-parameter - can be NULL. Returns the size of one FIFO entry in byte */
EXIMPORT RTK_ERROR
RtkGetPlainFifoInfo(RTK_PLAIN_FIFO_H hFifo, ULONG* lpulFifoFree, ULONG* lpulFifoUsed, ULONG* lpulFifoEntrySize);

#ifdef __cplusplus
}
#endif

#endif
```

#### rtkSemaphore.h
```c
/**
 * @file
 * @brief RTK semaphore functions
 *
 * Semaphores can be used to control access to critical code sections or to synchronize tasks.
 *
 * @ingroup rtk
 */

#ifndef _RTK_SEMAPHORE_H_
#define _RTK_SEMAPHORE_H_

#include <rtkBase.h>

#ifdef __cplusplus
extern "C" {
#endif

/** @brief RTK semaphore handle */
typedef RTK_H RTK_SEM_H;

/**
 * @brief Creates a semaphore with the provided name ('lpszSemaphoreName' must be unique or NULL).
 *
 * 'ulInitCount' defines the initial value of the semaphore (RtkAcquireSemaphore() decreases this value until 0,
 * RtkReleaseSemaphore() increases this value until 'ulMaxCount').
 * The output-parameter 'hSemaphore' (must not be NULL) returns a handle to the semaphore */
EXIMPORT RTK_ERROR
RtkCreateSemaphoreEx(const char* lpszSemaphoreName, ULONG ulInitCount, ULONG ulMaxCount, RTK_SEM_H* hSemaphore);

/**
 * @brief Creates a semaphore with the provided name ('lpszSemaphoreName' must be unique or NULL).
 *
 * The initial value of the semaphore is 'ulMaxCount' (RtkAcquireSemaphore() decreases this value until 0,
 * RtkReleaseSemaphore() increases this value until 'ulMaxCount').
 * The output-parameter 'hSemaphore' (must not be NULL) returns a handle to the semaphore */
EXIMPORT RTK_ERROR RtkCreateSemaphore(const char* lpszSemaphoreName, ULONG ulMaxCount, RTK_SEM_H* hSemaphore);

/**
 * @brief Deletes a sempahore */
EXIMPORT RTK_ERROR RtkDeleteSemaphore(RTK_SEM_H hSemaphore);

/**
 * @brief Blocks until the semaphore has a value higher than 0 or until the timeout expires.
 *
 * When the semaphore has a value higher than 0, then this function decrements this value and returns. */
EXIMPORT RTK_ERROR RtkAcquireSemaphore(RTK_SEM_H hSemaphore, ULONG ulTimeoutUsec);

/** @brief Increment the value of the semaphore.
 *
 *  Only if the value was lower than the 'ulMaxCount' defined when creating the semaphore. */
EXIMPORT RTK_ERROR RtkReleaseSemaphore(RTK_SEM_H hSemaphore);

/**
 * @brief Obtains information about the semaphore.
 * @param lpulMaxCount         Output-parameter - can be NULL. Returns ulMaxCount defined when creating the semaphore
 * @param lpulActCount         Output-parameter - can be NULL. Returns the current value of the semaphore
 * @param lpulTaskWaitingCount Output-parameter - can be NULL. Returns the number of tasks waiting for this semaphore */
EXIMPORT RTK_ERROR
RtkGetSemaphoreInfo(RTK_SEM_H hSemaphore, ULONG* lpulMaxCount, ULONG* lpulActCount, ULONG* lpulTaskWaitingCount);

#ifdef __cplusplus
}
#endif

#endif
```

#### rtkSharedMemory.h
```c
/**
 * @file
 * @brief RTK shared memory functions
 * @ingroup rtk
 */

#ifndef _RTK_SHARED_MEMORY_H_
#define _RTK_SHARED_MEMORY_H_

#include <rtkBase.h>

#ifdef __cplusplus
extern "C" {
#endif

/** @brief RTK shared memory handle */
typedef RTK_H RTK_SHARED_MEM_H;

/**
 * @brief Creates a shared memory object with the provided name ('lpszSharedMemoryName' must be unique or NULL).
 *
 * Allocates memory of size 'ulByteLength'.
 * A handle to the shared memory is returned as output-parameter ('hSharedMemory' - must not be NULL) */
EXIMPORT RTK_ERROR
RtkCreateSharedMemory(const char* lpszSharedMemoryName, ULONG ulByteLength, RTK_SHARED_MEM_H* hSharedMemory);

/** @brief Deletes a shared memory object */
EXIMPORT RTK_ERROR RtkDeleteSharedMemory(RTK_SHARED_MEM_H hSharedMemory);

/**
 * @brief Registers for usage of the shared memory.
 *
 * Obtains the memory address ('lpMemoryAddress' - must not be NULL) of the shared memory. Data can then be read/written
 * to this address. */
EXIMPORT RTK_ERROR RtkMapSharedMemory(RTK_SHARED_MEM_H hSharedMemory, void** lpMemoryAddress);

/**
 * @brief Unregisters usage of this shared memory. */
EXIMPORT RTK_ERROR RtkUnmapSharedMemory(RTK_SHARED_MEM_H hSharedMemory);

#ifdef __cplusplus
}
#endif

#endif
```

#### rtkBase.h
```c
/**
 * @file
 * @brief RTK basis data types and error codes
 * @ingroup rtk
 */

#ifndef _RTK_BASE_H_
#define _RTK_BASE_H_

#ifdef __cplusplus
extern "C" {
#endif

#include <rtkTypes.h>
#include <arexport.h>

/** @cond */

/* For using this file in Automation Studio tasks, it has to be included AFTER AsDefault.h */
#if defined (_DEFAULT_INCLUDES) && !defined(_RUNTIME_) && !defined(_REPLACE_CONST)
#error Rtk-headers have to be be included after AsDefault.h
#endif

/* COMPILER_SPECIFICS */
#ifndef DECLSPEC_NOTHROW
#if defined(__GNUC__) && ((__GNUC__ > 3) || ((__GNUC__ == 3) && (__GNUC_MINOR__ >= 3)))
#define DECLSPEC_NOTHROW __attribute__((__nothrow__))
#elif defined(__cplusplus) && (_MSC_VER >= 1200)
#define DECLSPEC_NOTHROW __declspec(nothrow)
#else
#define DECLSPEC_NOTHROW
#endif
#endif

/* Can be used to decorate RTK functions with additional attributes. */
#ifndef EXIMPORT
#if defined(_CPPUNWIND) || defined(__EXCEPTIONS)
#define EXIMPORT DECLSPEC_NOTHROW
#else
#define EXIMPORT
#endif
#endif

/** @endcond */

/** @name General definitions for RT kernel */
/*@{*/
/**
 * @brief Maximum length of an RTK object (task name, ...).
 * @note Longer names will be shortened to the maximum length! No error is reported. */
#define MAX_RTK_NAME_LENGTH 32
#define MAX_RTK_NAME_TERMINATED_LENGTH (MAX_RTK_NAME_LENGTH + 1)
/*@}*/

/** @name Timeout for task events, semaphore, fifo, debugmessage, ... */
/*@{*/
#define RTK_TIMEOUT_NOWAIT 0
#define RTK_TIMEOUT_WAITFOREVER 0xFFFFFFFF
/*@}*/

/** @brief RTK task function prototype */
typedef void (*LPRTK_CREATE_TASK_FKT)(void* param);

/**
 * @brief ERR_OK could be defined by spserror.h or runtime.h
 * @note If a stdlib has spserror.h included, we have to return ERR_OK 0U because the stdlibs catch ERR_OK with 0U via runtime.h */
#ifndef ERR_OK
#define ERR_OK 0U
#endif

/** @brief RTK error codes */
/* 25100 - 25199 obsolete (Debugger error codes) */
typedef enum
{
	ERR_RTK_OK = ERR_OK,

	ERR_RTK_OBJID = 25000, /**< @brief Invalid object ident */
	ERR_RTK_OBJNOTFOUND,   /**< @brief Object with specified name not found */
	ERR_RTK_OBJTYPE,       /**< @brief Invalid object type */
	ERR_RTK_OBJ_OVERFLOW,  /**< @brief Object table full */
	ERR_RTK_OBJ_EXIST,     /**< @brief Object already exists */
	ERR_RTK_OBJNAME,       /**< @brief Wrong object name */

	ERR_RTK_PRIORITY = 25010, /**< @brief Invalid priority */
	ERR_RTK_NO_STACK,         /**< @brief Not enough free stack */
	ERR_RTK_NOT_SUSPENDED,    /**< @brief Task is not suspended */
	ERR_RTK_SUSPENDED,        /**< @brief Task is already suspended */
	ERR_RTK_TASKVALUE,        /**< @brief Invalid valueindex */
	ERR_RTK_NOTASKTIMERS,     /**< @brief No more task timers available */
	ERR_RTK_TASKCREATE,       /**< @brief OS task not created */
	ERR_RTK_TASKDELETE,       /**< @brief OS Task not deleted */

	ERR_RTK_FIFO_CREATE = 25030,   /**< @brief FIFO not created (memory alloc, ...) */
	ERR_RTK_FIFO_DELETE,           /**< @brief FIFO not deleted (memory free, ...) */
	ERR_RTK_FIFO_WRITE,            /**< @brief FIFO not written (fifo full, ...) */
	ERR_RTK_FIFO_READ,             /**< @brief FIFO not read (fifo empty, ...) */
	ERR_RTK_FIFO_RELEASE,          /**< @brief FIFO not released */
	ERR_RTK_FIFO_ATTACHED_TIMEOUT, /**< @brief FIFO read/write with timeout invalid (attached) */
	ERR_RTK_FIFO_NOT_ATTACHED,     /**< @brief FIFO not attached when read/write */
	ERR_RTK_FIFO_ATTACHED,         /**< @brief FIFO already attached (other task) */
	ERR_RTK_FIFO_ATTACH,           /**< @brief FIFO not created for attach */

	ERR_RTK_SEMACREATE = 25040, /**< @brief OS semaphore not created */
	ERR_RTK_SEMA_DELETE,        /**< @brief OS semaphore not deleted */
	ERR_RTK_SEMA_RELEASE,       /**< @brief OS semaphore not released */

	ERR_WRONG_MEMTYPE = 25060, /**< @brief Invalid memory type */
	ERR_RTK_NOMEM_HEAP,        /**< @brief Not enough memory free in heap */
	ERR_RTK_FREE_HEAP,         /**< @brief Memory not in heap */

	ERR_RTK_CREATE_SHAREDMEM, /**< @brief SharedMemory not created */
	ERR_RTK_DELETE_SHAREDMEM, /**< @brief SharedMemory not deleted */
	ERR_RTK_MAP_SHAREDMEM,    /**< @brief SharedMemory not mapped */
	ERR_RTK_UNMAP_SHAREDMEM,  /**< @brief SharedMemory not unmapped */

	ERR_RTK_IRQNUMBER = 25080, /**< @brief Invalid interruptnumber */
	ERR_RTK_CONNECT_IRQ,       /**< @brief Interrupt not connected */
	ERR_RTK_DISCONNECT_IRQ,    /**< @brief Interrupt not disconnected */

	ERR_RTK_TIMERCYCLE = 25090, /**< @brief Invalid cycletime */
	ERR_RTK_WRONGTIME,          /**< @brief Invalid time/date */
	ERR_RTK_SET_RTC,            /**< @brief RealTimeClock not set */
	ERR_RTK_TIMER_CREATE,       /**< @brief Timer not created */
	ERR_RTK_TIMER_DELETE,       /**< @brief Timer not deleted */
	ERR_RTK_TIMER_START,        /**< @brief Timer not started */
	ERR_RTK_TIMER_STOP,         /**< @brief Timer not stopped */

	ERR_RTK_SOFTPLC_CREATE = 25200, /**< @brief RtkCreateSoftPlc not possible */
	ERR_RTK_INIT,                   /**< @brief RTK not initialized */
	ERR_RTK_DEINIT,                 /**< @brief RTK not deinitialized */
	ERR_RTK_FATAL,                  /**< @brief Fatal internal RTK error */
	ERR_RTK_TIMEOUT,                /**< @brief Timeout in RTK functions with wait */
	ERR_RTK_NOTSUPPORTED,           /**< @brief Function not supported in this RTK version */
	ERR_RTK_UNHANDLED_CPP_EXC,      /**< @brief Unhandled CPP Exception */

	ERR_RTK_CRITSECCREATE = 25250, /**< @brief CriticalSection not created */
	ERR_RTK_CRITSECDELETE,         /**< @brief CriticalSection not deleted */
	ERR_RTK_CRITSECENTER,          /**< @brief CriticalSection not enterd */
	ERR_RTK_CRITSECLEAVE,          /**< @brief CriticalSection not left */

	ERR_RTK_EXC_BASE = 25300, /**< @brief Base for RTK exceptions -> + RTK_EXCTYP_xx */

	ERR_RTK_LOG_CREATE = 25400, /**< @brief Log not created */
	ERR_RTK_LOG_DELETE,         /**< @brief Log not deleted  */
	ERR_RTK_LOG_NOBUFSET,       /**< @brief no Log-Buffer set */
	ERR_RTK_LOG_LOGACTIVE,      /**< @brief Log active */
} RTK_ERROR;

/** @brief General RTK object handle */
typedef ULONG RTK_H;

#ifdef __cplusplus
}
#endif

#endif
```

#### rtkCriticalSection.h
```c
/**
 * @file
 * @brief RTK critical section functions
 *
 * Critical Section
 * A critical section can be used to mutually exclude access to critical code sections which
 * process shared data that might be simultaneously modified by other tasks as well.
 * RTK critical sections support priority inheritance to avoid priority inversion.
 *
 * @ingroup rtk
 */

#ifndef _RTK_CRITICAL_SECTION_H_
#define _RTK_CRITICAL_SECTION_H_

#include <rtkBase.h>

#ifdef __cplusplus
extern "C" {
#endif

/** @brief RTK critical section handle */
typedef RTK_H RTK_CRIT_SEC_H;

/**
 * @brief Creates a critical section object with the provided name ('lpszCriticalSectionName' must be unique or NULL).
 *
 * The output-parameter 'hCriticalSection' (must not be NULL) returns a handle to the critical section */
EXIMPORT RTK_ERROR RtkCreateCriticalSection(const char* lpszCriticalSectionName, RTK_CRIT_SEC_H* hCriticalSection);

/** @brief Deletes a critical section object. */
EXIMPORT RTK_ERROR RtkDeleteCriticalSection(RTK_CRIT_SEC_H hCriticalSection);

/**
 * @brief Enter a critical section.
 *
 * This function has to be called before accessing the data which needs mutual exclusion.
 * If no other task is in the critical section (entered and did not yet leave), then this function returns immediately.
 * If another task is in the critical section, then the current task yields until no other
 * task is in the critical section. */
EXIMPORT RTK_ERROR RtkEnterCriticalSection(RTK_CRIT_SEC_H hCriticalSection);

/**
 * @brief Leave a critical section.
 *
 * This function has to be called after accessing the data which needs mutual exclusion. */
EXIMPORT RTK_ERROR RtkLeaveCriticalSection(RTK_CRIT_SEC_H hCriticalSection);

#ifdef __cplusplus
}
#endif

#endif
```

#### rtkFifo.h
```c
/**
 * @file
 * @brief RTK FIFO functions
 * @ingroup rtk
 */

#ifndef _RTK_FIFO_H_
#define _RTK_FIFO_H_

#include <rtkBase.h>

#ifdef __cplusplus
extern "C" {
#endif

/** @brief RTK FIFO handle */
typedef RTK_H RTK_FIFO_H;

/** @brief Type of FIFO flags */
typedef unsigned long RTK_FIFOFLAG;

/** @name Fifo flags (create) */
/*@{*/
#define RTK_FIFO_WRITE_UNTIL_FULL 0x00000000 /**< @brief no overwrite */
#define RTK_FIFO_WRITE_ALWAYS 0x00000001     /**< @brief overwrite */
#define RTK_FIFO_ATTACH 0x00000002           /**< @brief FIFO access only attach/release */
/*@}*/

/**
 * @brief Creates a FIFO with the provided name ('lpszFifoName' must be unique or NULL) and the provided size ('ulFifoByteSize').
 *
 * The 'FifoFlags' determine whether RtkWriteFifo calls will overwrite data in the FIFO (#RTK_FIFO_WRITE_ALWAYS) or whether
 * RtkWriteFifo calls only succeed if there is enough free space available in the FIFO (#RTK_FIFO_WRITE_UNTIL_FULL).
 * A handle to the FIFO is returned as output-parameter ('hFifo' - must not be NULL) */
EXIMPORT RTK_ERROR
RtkCreateFifo(const char* lpszFifoName, ULONG ulFifoByteSize, RTK_FIFOFLAG FifoFlags, RTK_FIFO_H* hFifo);

/** @brief Deletes a FIFO. */
EXIMPORT RTK_ERROR RtkDeleteFifo(RTK_FIFO_H hFifo);

/**
 * @brief Writes data ('lpDataSource') with size 'ulDataByteSize' to the FIFO.
 *
 * If the FIFO was created with the flag #RTK_FIFO_WRITE_ALWAYS, then unread data will be overwritten.
 * If the FIFO was created with the flag #RTK_FIFO_WRITE_UNTIL_FULL, then unread data will not be overwritten and this
 * function waits for 'ulTimeoutUsec' (RTK_TIMEOUT_WAITFOREVER to wait forever) to put the data into the FIFO and
 * returns #ERR_RTK_TIMEOUT if the timeout expires. */
EXIMPORT RTK_ERROR RtkWriteFifo(RTK_FIFO_H hFifo, const void* lpDataSource, ULONG ulDataByteSize, ULONG ulTimeoutUsec);

/**
 * @brief Copies data of size 'lpDataByteSize' from the FIFO to 'lpDataDest' (must not be NULL).
 *
 * Waits for 'ulTimeoutUsec' (RTK_TIMEOUT_WAITFOREVER to wait forever) if not enough data is available in the FIFO. */
EXIMPORT RTK_ERROR RtkReadFifo(RTK_FIFO_H hFifo, void* lpDataDest, ULONG lpDataByteSize, ULONG ulTimeoutUsec);

/**
 * @brief Deletes all data in the FIFO. */
EXIMPORT RTK_ERROR RtkClearFifo(RTK_FIFO_H hFifo);

/**
 * @brief Locks access (read/write) to the FIFO for other tasks.
 *
 * It is possible to have one task reading and one task writing to the FIFO without requiring locking with this
 * function. However, if multiple tasks read or if multiple tasks write to the FIFO, then locking with this function is
 * required. */
EXIMPORT RTK_ERROR RtkAttachFifo(RTK_FIFO_H hFifo);

/** @brief Unlocks access (read/write) to the FIFO for other tasks. */
EXIMPORT RTK_ERROR RtkReleaseFifo(RTK_FIFO_H hFifo);

/**
 * @brief Obtains information about the FIFO.
 * @param hFifo        Handle to the FIFO for which the information shall be retrieved.
 * @param lpulFifoFree Output-parameter - can be NULL. Returns the number of free bytes.
 * @param lpulFifoUsed Output-parameter - can be NULL. Returns the number of occupied bytes. */
EXIMPORT RTK_ERROR RtkGetFifoInfo(RTK_FIFO_H hFifo, ULONG* lpulFifoFree, ULONG* lpulFifoUsed);

#ifdef __cplusplus
}
#endif

#endif
```

#### rtkInterrupt.h
```c
/**
 * @file
 * @brief RTK interrupt functions
 * @ingroup rtk
 * @note Do not use this interface!
 */

#ifndef _RTK_INTERRUPT_H_
#define _RTK_INTERRUPT_H_

#include <arexport.h>

#ifdef __cplusplus
extern "C" {
#endif

/** @brief Disables all interrupts */
AR_NOT_RECOMMENDED void RtkDisableInterrupts(void);

/** @brief Re-enables interrupts which were disabled by calling RtkDisableInterrupts */
AR_NOT_RECOMMENDED void RtkEnableInterrupts(void);

#ifdef __cplusplus
}
#endif

#endif
```
